ABB RAPID module: 3c2a8035.mod

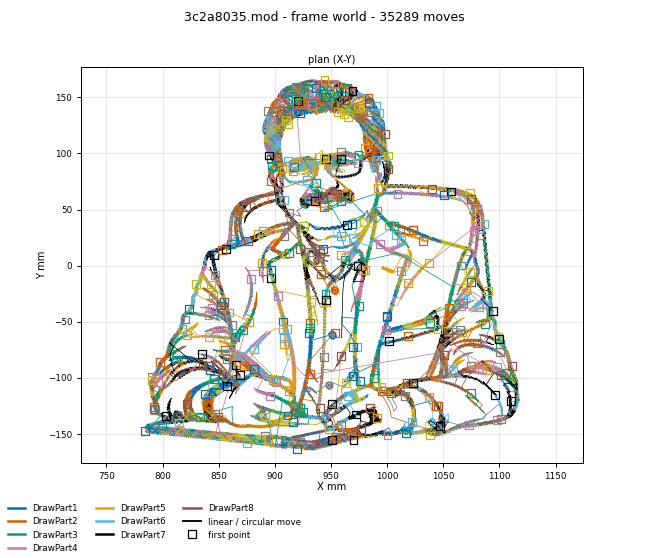
[picture p0: tool path of 3c2a8035.mod in frame world, 35289 of 35291 moves have a stored position in this frame; points joined in program order, loops and branches not executed]
MODULE ImageDraw
  ! Generated 2026-10-07 06:23 for ABB IRB 1600-10/1.45: 2961 strokes
  ! Page 500 x 350 mm. Work object wPaper: Z points up, so pen-up is +Z and the tool uses orientation [0,1,0,0].
  PERS tooldata tPen:=[TRUE,[[0,0,120],[1,0,0,0]],[0.3,[0,0,60],[1,0,0,0],0,0,0]];
  PERS wobjdata wPaper:=[FALSE,TRUE,"",[[700,-175,0],[1,0,0,0]],[[0,0,0],[1,0,0,0]]];
  CONST robtarget pOrigin:=[[0,0,0],[0,1,0,0],[0,0,0,0],[9E9,9E9,9E9,9E9,9E9,9E9]];
  CONST jointtarget jHome:=[[0,0,0,0,30,0],[9E9,9E9,9E9,9E9,9E9,9E9]];
  CONST speeddata vTravel:=[250,200,5000,1000];

  PROC DrawImage()
    SingArea\Wrist;
    ConfL\Off;
    ConfJ\Off;
    MoveAbsJ jHome\NoEOffs,vTravel,fine,tPen;
    DrawPart1;
    DrawPart2;
    DrawPart3;
    DrawPart4;
    DrawPart5;
    DrawPart6;
    DrawPart7;
    DrawPart8;
    DrawPart9;
    DrawPart10;
    DrawPart11;
    DrawPart12;
    DrawPart13;
    DrawPart14;
    DrawPart15;
    DrawPart16;
    DrawPart17;
    DrawPart18;
    DrawPart19;
    DrawPart20;
    DrawPart21;
    DrawPart22;
    DrawPart23;
    DrawPart24;
    DrawPart25;
    DrawPart26;
    DrawPart27;
    DrawPart28;
    DrawPart29;
    DrawPart30;
    DrawPart31;
    DrawPart32;
    DrawPart33;
    DrawPart34;
    DrawPart35;
    DrawPart36;
    DrawPart37;
    DrawPart38;
    DrawPart39;
    DrawPart40;
    DrawPart41;
    DrawPart42;
    DrawPart43;
    DrawPart44;
    DrawPart45;
    DrawPart46;
    DrawPart47;
    DrawPart48;
    DrawPart49;
    DrawPart50;
    DrawPart51;
    DrawPart52;
    DrawPart53;
    DrawPart54;
    DrawPart55;
    DrawPart56;
    DrawPart57;
    DrawPart58;
    DrawPart59;
    DrawPart60;
    DrawPart61;
    DrawPart62;
    DrawPart63;
    DrawPart64;
    DrawPart65;
    DrawPart66;
    DrawPart67;
    DrawPart68;
    DrawPart69;
    DrawPart70;
    DrawPart71;
    DrawPart72;
    DrawPart73;
    DrawPart74;
    DrawPart75;
    DrawPart76;
    DrawPart77;
    DrawPart78;
    DrawPart79;
    DrawPart80;
    DrawPart81;
    DrawPart82;
    DrawPart83;
    DrawPart84;
    DrawPart85;
    DrawPart86;
    DrawPart87;
    DrawPart88;
    DrawPart89;
    DrawPart90;
    DrawPart91;
    DrawPart92;
    DrawPart93;
    DrawPart94;
    DrawPart95;
    DrawPart96;
    DrawPart97;
    DrawPart98;
    DrawPart99;
    DrawPart100;
    DrawPart101;
    DrawPart102;
    DrawPart103;
    DrawPart104;
    DrawPart105;
    DrawPart106;
    DrawPart107;
    DrawPart108;
    DrawPart109;
    DrawPart110;
    DrawPart111;
    DrawPart112;
    DrawPart113;
    DrawPart114;
    DrawPart115;
    DrawPart116;
    DrawPart117;
    DrawPart118;
    DrawPart119;
    DrawPart120;
    DrawPart121;
    DrawPart122;
    DrawPart123;
    DrawPart124;
    DrawPart125;
    DrawPart126;
    DrawPart127;
    DrawPart128;
    DrawPart129;
    DrawPart130;
    DrawPart131;
    DrawPart132;
    DrawPart133;
    DrawPart134;
    DrawPart135;
    DrawPart136;
    DrawPart137;
    DrawPart138;
    DrawPart139;
    DrawPart140;
    DrawPart141;
    DrawPart142;
    DrawPart143;
    DrawPart144;
    DrawPart145;
    DrawPart146;
    DrawPart147;
    DrawPart148;
    DrawPart149;
    DrawPart150;
    DrawPart151;
    DrawPart152;
    DrawPart153;
    DrawPart154;
    DrawPart155;
    DrawPart156;
    DrawPart157;
    DrawPart158;
    DrawPart159;
    DrawPart160;
    DrawPart161;
    DrawPart162;
    DrawPart163;
    DrawPart164;
    DrawPart165;
    DrawPart166;
    DrawPart167;
    DrawPart168;
    DrawPart169;
    DrawPart170;
    DrawPart171;
    DrawPart172;
    DrawPart173;
    DrawPart174;
    DrawPart175;
    DrawPart176;
    DrawPart177;
    DrawPart178;
    DrawPart179;
    DrawPart180;
    DrawPart181;
    DrawPart182;
    DrawPart183;
    DrawPart184;
    DrawPart185;
    DrawPart186;
    DrawPart187;
    DrawPart188;
    DrawPart189;
    DrawPart190;
    DrawPart191;
    DrawPart192;
    DrawPart193;
    DrawPart194;
    DrawPart195;
    DrawPart196;
    DrawPart197;
    DrawPart198;
    DrawPart199;
    DrawPart200;
    DrawPart201;
    DrawPart202;
    DrawPart203;
    DrawPart204;
    DrawPart205;
    DrawPart206;
    DrawPart207;
    DrawPart208;
    DrawPart209;
    DrawPart210;
    DrawPart211;
    DrawPart212;
    DrawPart213;
    DrawPart214;
    DrawPart215;
    DrawPart216;
    DrawPart217;
    DrawPart218;
    DrawPart219;
    DrawPart220;
    DrawPart221;
    DrawPart222;
    DrawPart223;
    DrawPart224;
    DrawPart225;
    DrawPart226;
    DrawPart227;
    DrawPart228;
    DrawPart229;
    DrawPart230;
    DrawPart231;
    DrawPart232;
    DrawPart233;
    DrawPart234;
    DrawPart235;
    DrawPart236;
    DrawPart237;
    DrawPart238;
    DrawPart239;
    DrawPart240;
    DrawPart241;
    DrawPart242;
    DrawPart243;
    DrawPart244;
    DrawPart245;
    DrawPart246;
    DrawPart247;
    DrawPart248;
    DrawPart249;
    DrawPart250;
    DrawPart251;
    DrawPart252;
    DrawPart253;
    DrawPart254;
    DrawPart255;
    DrawPart256;
    DrawPart257;
    DrawPart258;
    DrawPart259;
    DrawPart260;
    DrawPart261;
    DrawPart262;
    DrawPart263;
    DrawPart264;
    DrawPart265;
    DrawPart266;
    DrawPart267;
    DrawPart268;
    DrawPart269;
    DrawPart270;
    DrawPart271;
    DrawPart272;
    DrawPart273;
    DrawPart274;
    DrawPart275;
    DrawPart276;
    DrawPart277;
    DrawPart278;
    DrawPart279;
    DrawPart280;
    DrawPart281;
    DrawPart282;
    DrawPart283;
    DrawPart284;
    DrawPart285;
    DrawPart286;
    DrawPart287;
    DrawPart288;
    DrawPart289;
    DrawPart290;
    DrawPart291;
    DrawPart292;
    DrawPart293;
    DrawPart294;
    DrawPart295;
    MoveAbsJ jHome\NoEOffs,vTravel,fine,tPen;
  ENDPROC

  PROC DrawPart1()
    MoveL Offs(pOrigin,84.39,27.87,6.00),vTravel,z5,tPen\WObj:=wPaper;
    MoveL Offs(pOrigin,84.39,27.87,0.00),v60,z0,tPen\WObj:=wPaper;
    MoveL Offs(pOrigin,86.34,25.92,0.00),v40,z0,tPen\WObj:=wPaper;
    MoveL Offs(pOrigin,86.59,26.62,0.00),v40,z0,tPen\WObj:=wPaper;
    MoveL Offs(pOrigin,99.12,26.62,0.00),v40,fine,tPen\WObj:=wPaper;
    MoveL Offs(pOrigin,99.12,26.62,6.00),v60,z5,tPen\WObj:=wPaper;
    MoveL Offs(pOrigin,99.50,25.13,6.00),vTravel,z5,tPen\WObj:=wPaper;
    MoveL Offs(pOrigin,99.50,25.13,0.00),v60,z0,tPen\WObj:=wPaper;
    MoveL Offs(pOrigin,105.21,30.84,0.00),v40,z0,tPen\WObj:=wPaper;
    MoveL Offs(pOrigin,104.60,31.55,0.00),v40,z0,tPen\WObj:=wPaper;
    MoveL Offs(pOrigin,113.01,23.14,0.00),v40,z0,tPen\WObj:=wPaper;
    MoveL Offs(pOrigin,113.13,23.82,0.00),v40,z0,tPen\WObj:=wPaper;
    MoveL Offs(pOrigin,118.84,29.53,0.00),v40,z0,tPen\WObj:=wPaper;
    MoveL Offs(pOrigin,119.58,30.01,0.00),v40,z0,tPen\WObj:=wPaper;
    MoveL Offs(pOrigin,128.15,21.44,0.00),v40,z0,tPen\WObj:=wPaper;
    MoveL Offs(pOrigin,127.96,22.22,0.00),v40,z0,tPen\WObj:=wPaper;
    MoveL Offs(pOrigin,129.76,24.02,0.00),v40,z0,tPen\WObj:=wPaper;
    MoveL Offs(pOrigin,129.72,23.45,0.00),v40,z0,tPen\WObj:=wPaper;
    MoveL Offs(pOrigin,117.19,23.45,0.00),v40,z0,tPen\WObj:=wPaper;
    MoveL Offs(pOrigin,117.17,23.38,0.00),v40,z0,tPen\WObj:=wPaper;
    MoveL Offs(pOrigin,118.98,25.19,0.00),v40,z0,tPen\WObj:=wPaper;
    MoveL Offs(pOrigin,119.74,24.50,0.00),v40,z0,tPen\WObj:=wPaper;
    MoveL Offs(pOrigin,107.62,24.50,0.00),v40,z0,tPen\WObj:=wPaper;
    MoveL Offs(pOrigin,107.74,24.40,0.00),v40,z0,tPen\WObj:=wPaper;
    MoveL Offs(pOrigin,113.30,29.96,0.00),v40,z0,tPen\WObj:=wPaper;
    MoveL Offs(pOrigin,112.99,30.63,0.00),v40,z0,tPen\WObj:=wPaper;
    MoveL Offs(pOrigin,121.40,22.21,0.00),v40,z0,tPen\WObj:=wPaper;
    MoveL Offs(pOrigin,121.07,22.80,0.00),v40,z0,tPen\WObj:=wPaper;
    MoveL Offs(pOrigin,126.93,28.66,0.00),v40,z0,tPen\WObj:=wPaper;
    MoveL Offs(pOrigin,126.18,29.39,0.00),v40,z0,tPen\WObj:=wPaper;
    MoveL Offs(pOrigin,134.74,20.82,0.00),v40,z0,tPen\WObj:=wPaper;
    MoveL Offs(pOrigin,134.70,21.49,0.00),v40,z0,tPen\WObj:=wPaper;
    MoveL Offs(pOrigin,136.50,23.29,0.00),v40,z0,tPen\WObj:=wPaper;
    MoveL Offs(pOrigin,135.90,24.19,0.00),v40,z0,tPen\WObj:=wPaper;
    MoveL Offs(pOrigin,139.21,27.50,0.00),v40,z0,tPen\WObj:=wPaper;
    MoveL Offs(pOrigin,139.36,28.15,0.00),v40,z0,tPen\WObj:=wPaper;
    MoveL Offs(pOrigin,148.08,19.43,0.00),v40,z0,tPen\WObj:=wPaper;
    MoveL Offs(pOrigin,148.32,20.18,0.00),v40,z0,tPen\WObj:=wPaper;
    MoveL Offs(pOrigin,150.13,21.99,0.00),v40,z0,tPen\WObj:=wPaper;
    MoveL Offs(pOrigin,150.55,21.34,0.00),v40,z0,tPen\WObj:=wPaper;
    MoveL Offs(pOrigin,138.65,21.34,0.00),v40,z0,tPen\WObj:=wPaper;
    MoveL Offs(pOrigin,138.89,21.20,0.00),v40,z0,tPen\WObj:=wPaper;
    MoveL Offs(pOrigin,140.54,22.86,0.00),v40,z0,tPen\WObj:=wPaper;
    MoveL Offs(pOrigin,139.95,23.75,0.00),v40,z0,tPen\WObj:=wPaper;
    MoveL Offs(pOrigin,141.75,25.56,0.00),v40,z0,tPen\WObj:=wPaper;
    MoveL Offs(pOrigin,142.50,26.31,0.00),v40,z0,tPen\WObj:=wPaper;
    MoveL Offs(pOrigin,143.25,27.06,0.00),v40,z0,tPen\WObj:=wPaper;
    MoveL Offs(pOrigin,142.81,27.69,0.00),v40,z0,tPen\WObj:=wPaper;
    MoveL Offs(pOrigin,151.37,19.12,0.00),v40,z0,tPen\WObj:=wPaper;
    MoveL Offs(pOrigin,151.02,19.89,0.00),v40,z0,tPen\WObj:=wPaper;
    MoveL Offs(pOrigin,157.03,25.90,0.00),v40,z0,tPen\WObj:=wPaper;
    MoveL Offs(pOrigin,157.49,26.45,0.00),v40,z0,tPen\WObj:=wPaper;
    MoveL Offs(pOrigin,166.51,17.43,0.00),v40,z0,tPen\WObj:=wPaper;
    MoveL Offs(pOrigin,167.04,17.99,0.00),v40,z0,tPen\WObj:=wPaper;
    MoveL Offs(pOrigin,171.10,22.05,0.00),v40,z0,tPen\WObj:=wPaper;
    MoveL Offs(pOrigin,171.80,21.34,0.00),v40,z0,tPen\WObj:=wPaper;
    MoveL Offs(pOrigin,168.19,21.34,0.00),v40,z0,tPen\WObj:=wPaper;
    MoveL Offs(pOrigin,168.25,22.19,0.00),v40,z0,tPen\WObj:=wPaper;
    MoveL Offs(pOrigin,164.50,18.43,0.00),v40,z0,tPen\WObj:=wPaper;
    MoveL Offs(pOrigin,164.86,17.58,0.00),v40,z0,tPen\WObj:=wPaper;
    MoveL Offs(pOrigin,155.84,26.60,0.00),v40,z0,tPen\WObj:=wPaper;
    MoveL Offs(pOrigin,155.83,26.20,0.00),v40,z0,tPen\WObj:=wPaper;
    MoveL Offs(pOrigin,152.07,22.44,0.00),v40,z0,tPen\WObj:=wPaper;
    MoveL Offs(pOrigin,151.32,21.69,0.00),v40,z0,tPen\WObj:=wPaper;
    MoveL Offs(pOrigin,149.52,19.89,0.00),v40,z0,tPen\WObj:=wPaper;
    MoveL Offs(pOrigin,149.57,19.43,0.00),v40,z0,tPen\WObj:=wPaper;
    MoveL Offs(pOrigin,141.01,27.99,0.00),v40,z0,tPen\WObj:=wPaper;
    MoveL Offs(pOrigin,140.56,27.35,0.00),v40,z0,tPen\WObj:=wPaper;
    MoveL Offs(pOrigin,137.40,24.19,0.00),v40,z0,tPen\WObj:=wPaper;
    MoveL Offs(pOrigin,137.85,23.15,0.00),v40,z0,tPen\WObj:=wPaper;
    MoveL Offs(pOrigin,136.04,21.34,0.00),v40,z0,tPen\WObj:=wPaper;
    MoveL Offs(pOrigin,136.39,20.67,0.00),v40,z0,tPen\WObj:=wPaper;
    MoveL Offs(pOrigin,127.82,29.23,0.00),v40,z0,tPen\WObj:=wPaper;
    MoveL Offs(pOrigin,128.28,28.51,0.00),v40,z0,tPen\WObj:=wPaper;
    MoveL Offs(pOrigin,122.57,22.80,0.00),v40,z0,tPen\WObj:=wPaper;
    MoveL Offs(pOrigin,123.05,22.06,0.00),v40,z0,tPen\WObj:=wPaper;
    MoveL Offs(pOrigin,114.64,30.47,0.00),v40,z0,tPen\WObj:=wPaper;
    MoveL Offs(pOrigin,114.65,29.82,0.00),v40,z0,tPen\WObj:=wPaper;
    MoveL Offs(pOrigin,109.09,24.26,0.00),v40,fine,tPen\WObj:=wPaper;
    MoveL Offs(pOrigin,109.09,24.26,6.00),v60,z5,tPen\WObj:=wPaper;
    MoveL Offs(pOrigin,108.07,23.60,6.00),vTravel,z5,tPen\WObj:=wPaper;
    MoveL Offs(pOrigin,108.07,23.60,0.00),v60,z0,tPen\WObj:=wPaper;
    MoveL Offs(pOrigin,99.80,31.87,0.00),v40,z0,tPen\WObj:=wPaper;
    MoveL Offs(pOrigin,99.67,31.27,0.00),v40,z0,tPen\WObj:=wPaper;
    MoveL Offs(pOrigin,94.11,25.71,0.00),v40,z0,tPen\WObj:=wPaper;
    MoveL Offs(pOrigin,94.88,24.84,0.00),v40,z0,tPen\WObj:=wPaper;
    MoveL Offs(pOrigin,86.02,33.71,0.00),v40,z0,tPen\WObj:=wPaper;
    MoveL Offs(pOrigin,86.59,32.95,0.00),v40,z0,tPen\WObj:=wPaper;
    MoveL Offs(pOrigin,91.05,32.95,0.00),v40,z0,tPen\WObj:=wPaper;
    MoveL Offs(pOrigin,91.89,32.44,0.00),v40,z0,tPen\WObj:=wPaper;
    MoveL Offs(pOrigin,86.18,26.73,0.00),v40,z0,tPen\WObj:=wPaper;
    MoveL Offs(pOrigin,85.74,26.67,0.00),v40,z0,tPen\WObj:=wPaper;
    MoveL Offs(pOrigin,85.31,27.10,0.00),v40,z0,tPen\WObj:=wPaper;
    MoveL Offs(pOrigin,85.74,26.67,0.00),v40,z0,tPen\WObj:=wPaper;
    MoveL Offs(pOrigin,85.28,27.33,0.00),v40,z0,tPen\WObj:=wPaper;
    MoveL Offs(pOrigin,93.39,35.44,0.00),v40,z0,tPen\WObj:=wPaper;
    MoveL Offs(pOrigin,92.90,35.78,0.00),v40,z0,tPen\WObj:=wPaper;
    MoveL Offs(pOrigin,95.30,33.38,0.00),v40,z0,tPen\WObj:=wPaper;
    MoveL Offs(pOrigin,95.04,34.10,0.00),v40,z0,tPen\WObj:=wPaper;
    MoveL Offs(pOrigin,97.29,36.35,0.00),v40,z0,tPen\WObj:=wPaper;
    MoveL Offs(pOrigin,97.84,36.82,0.00),v40,z0,tPen\WObj:=wPaper;
    MoveL Offs(pOrigin,101.15,33.51,0.00),v40,fine,tPen\WObj:=wPaper;
    MoveL Offs(pOrigin,101.15,33.51,6.00),v60,z5,tPen\WObj:=wPaper;
    MoveL Offs(pOrigin,102.34,33.81,6.00),vTravel,z5,tPen\WObj:=wPaper;
    MoveL Offs(pOrigin,102.34,33.81,0.00),v60,z0,tPen\WObj:=wPaper;
    MoveL Offs(pOrigin,98.89,37.26,0.00),v40,z0,tPen\WObj:=wPaper;
    MoveL Offs(pOrigin,99.39,36.96,0.00),v40,z0,tPen\WObj:=wPaper;
    MoveL Offs(pOrigin,96.99,34.56,0.00),v40,z0,tPen\WObj:=wPaper;
    MoveL Offs(pOrigin,96.65,33.52,0.00),v40,z0,tPen\WObj:=wPaper;
    MoveL Offs(pOrigin,94.25,35.93,0.00),v40,z0,tPen\WObj:=wPaper;
    MoveL Offs(pOrigin,94.24,35.06,0.00),v40,z0,tPen\WObj:=wPaper;
    MoveL Offs(pOrigin,98.28,35.06,0.00),v40,z0,tPen\WObj:=wPaper;
    MoveL Offs(pOrigin,98.63,34.71,0.00),v40,z0,tPen\WObj:=wPaper;
    MoveL Offs(pOrigin,101.34,37.42,0.00),v40,z0,tPen\WObj:=wPaper;
    MoveL Offs(pOrigin,101.28,37.85,0.00),v40,z0,tPen\WObj:=wPaper;
    MoveL Offs(pOrigin,105.19,33.95,0.00),v40,fine,tPen\WObj:=wPaper;
    MoveL Offs(pOrigin,105.19,33.95,6.00),v60,z5,tPen\WObj:=wPaper;
    MoveL Offs(pOrigin,106.39,34.24,6.00),vTravel,z5,tPen\WObj:=wPaper;
    MoveL Offs(pOrigin,106.39,34.24,0.00),v60,z0,tPen\WObj:=wPaper;
    MoveL Offs(pOrigin,91.51,49.12,0.00),v40,z0,tPen\WObj:=wPaper;
  ENDPROC

  PROC DrawPart2()
    MoveL Offs(pOrigin,91.94,48.92,0.00),v40,z0,tPen\WObj:=wPaper;
    MoveL Offs(pOrigin,94.79,51.78,0.00),v40,z0,tPen\WObj:=wPaper;
    MoveL Offs(pOrigin,94.45,51.96,0.00),v40,z0,tPen\WObj:=wPaper;
    MoveL Offs(pOrigin,92.32,51.96,0.00),v40,z0,tPen\WObj:=wPaper;
    MoveL Offs(pOrigin,91.95,51.92,0.00),v40,z0,tPen\WObj:=wPaper;
    MoveL Offs(pOrigin,96.30,56.27,0.00),v40,z0,tPen\WObj:=wPaper;
    MoveL Offs(pOrigin,95.94,56.21,0.00),v40,z0,tPen\WObj:=wPaper;
    MoveL Offs(pOrigin,96.43,57.91,0.00),v40,z0,tPen\WObj:=wPaper;
    MoveL Offs(pOrigin,97.35,58.76,0.00),v40,z0,tPen\WObj:=wPaper;
    MoveL Offs(pOrigin,97.35,59.83,0.00),v40,z0,tPen\WObj:=wPaper;
    MoveL Offs(pOrigin,99.20,63.44,0.00),v40,z0,tPen\WObj:=wPaper;
    MoveL Offs(pOrigin,100.12,64.07,0.00),v40,z0,tPen\WObj:=wPaper;
    MoveL Offs(pOrigin,100.40,65.56,0.00),v40,z0,tPen\WObj:=wPaper;
    MoveL Offs(pOrigin,100.40,65.56,0.00),v40,z0,tPen\WObj:=wPaper;
    MoveL Offs(pOrigin,100.40,66.41,0.00),v40,z0,tPen\WObj:=wPaper;
    MoveL Offs(pOrigin,101.32,68.75,0.00),v40,z0,tPen\WObj:=wPaper;
    MoveL Offs(pOrigin,103.94,73.85,0.00),v40,z0,tPen\WObj:=wPaper;
    MoveL Offs(pOrigin,108.69,80.44,0.00),v40,z0,tPen\WObj:=wPaper;
    MoveL Offs(pOrigin,111.88,83.62,0.00),v40,z0,tPen\WObj:=wPaper;
    MoveL Offs(pOrigin,115.70,86.46,0.00),v40,z0,tPen\WObj:=wPaper;
    MoveL Offs(pOrigin,118.25,87.73,0.00),v40,z0,tPen\WObj:=wPaper;
    MoveL Offs(pOrigin,118.75,88.44,0.00),v40,z0,tPen\WObj:=wPaper;
    MoveL Offs(pOrigin,121.86,89.57,0.00),v40,z0,tPen\WObj:=wPaper;
    MoveL Offs(pOrigin,124.84,90.00,0.00),v40,z0,tPen\WObj:=wPaper;
    MoveL Offs(pOrigin,124.84,90.00,0.00),v40,z0,tPen\WObj:=wPaper;
    MoveL Offs(pOrigin,126.96,90.21,0.00),v40,z0,tPen\WObj:=wPaper;
    MoveL Offs(pOrigin,127.18,90.00,0.00),v40,z0,tPen\WObj:=wPaper;
    MoveL Offs(pOrigin,127.18,90.00,0.00),v40,z0,tPen\WObj:=wPaper;
    MoveL Offs(pOrigin,126.54,89.36,0.00),v40,z0,tPen\WObj:=wPaper;
    MoveL Offs(pOrigin,124.84,89.36,0.00),v40,z0,tPen\WObj:=wPaper;
    MoveL Offs(pOrigin,124.84,89.36,0.00),v40,z0,tPen\WObj:=wPaper;
    MoveL Offs(pOrigin,118.46,87.66,0.00),v40,z0,tPen\WObj:=wPaper;
    MoveL Offs(pOrigin,118.12,87.05,0.00),v40,z0,tPen\WObj:=wPaper;
    MoveL Offs(pOrigin,120.82,89.76,0.00),v40,z0,tPen\WObj:=wPaper;
    MoveL Offs(pOrigin,120.75,90.07,0.00),v40,z0,tPen\WObj:=wPaper;
    MoveL Offs(pOrigin,122.85,87.97,0.00),v40,z0,tPen\WObj:=wPaper;
    MoveL Offs(pOrigin,122.62,88.56,0.00),v40,z0,tPen\WObj:=wPaper;
    MoveL Offs(pOrigin,127.13,93.07,0.00),v40,z0,tPen\WObj:=wPaper;
    MoveL Offs(pOrigin,127.63,93.65,0.00),v40,z0,tPen\WObj:=wPaper;
    MoveL Offs(pOrigin,140.10,81.18,0.00),v40,z0,tPen\WObj:=wPaper;
    MoveL Offs(pOrigin,139.82,81.87,0.00),v40,z0,tPen\WObj:=wPaper;
    MoveL Offs(pOrigin,143.13,85.18,0.00),v40,z0,tPen\WObj:=wPaper;
    MoveL Offs(pOrigin,142.69,84.70,0.00),v40,z0,tPen\WObj:=wPaper;
    MoveL Offs(pOrigin,138.65,84.70,0.00),v40,z0,tPen\WObj:=wPaper;
    MoveL Offs(pOrigin,139.07,85.32,0.00),v40,z0,tPen\WObj:=wPaper;
    MoveL Offs(pOrigin,139.50,84.47,0.00),v40,z0,tPen\WObj:=wPaper;
    MoveL Offs(pOrigin,140.77,83.84,0.00),v40,z0,tPen\WObj:=wPaper;
    MoveL Offs(pOrigin,140.99,83.41,0.00),v40,z0,tPen\WObj:=wPaper;
    MoveL Offs(pOrigin,140.99,83.41,0.00),v40,z0,tPen\WObj:=wPaper;
    MoveL Offs(pOrigin,140.35,83.20,0.00),v40,z0,tPen\WObj:=wPaper;
    MoveL Offs(pOrigin,132.91,84.26,0.00),v40,z0,tPen\WObj:=wPaper;
    MoveL Offs(pOrigin,126.96,84.05,0.00),v40,z0,tPen\WObj:=wPaper;
    MoveL Offs(pOrigin,121.65,82.99,0.00),v40,z0,tPen\WObj:=wPaper;
    MoveL Offs(pOrigin,117.40,81.29,0.00),v40,z0,tPen\WObj:=wPaper;
    MoveL Offs(pOrigin,117.26,80.86,0.00),v40,z0,tPen\WObj:=wPaper;
    MoveL Offs(pOrigin,117.82,80.65,0.00),v40,z0,tPen\WObj:=wPaper;
    MoveL Offs(pOrigin,123.78,82.56,0.00),v40,z0,tPen\WObj:=wPaper;
    MoveL Offs(pOrigin,125.26,82.78,0.00),v40,z0,tPen\WObj:=wPaper;
    MoveL Offs(pOrigin,125.90,82.35,0.00),v40,z0,tPen\WObj:=wPaper;
    MoveL Offs(pOrigin,125.90,82.35,0.00),v40,z0,tPen\WObj:=wPaper;
    MoveL Offs(pOrigin,127.60,82.56,0.00),v40,z0,tPen\WObj:=wPaper;
    MoveL Offs(pOrigin,128.24,83.13,0.00),v40,z0,tPen\WObj:=wPaper;
    MoveL Offs(pOrigin,128.88,83.20,0.00),v40,z0,tPen\WObj:=wPaper;
    MoveL Offs(pOrigin,128.02,82.56,0.00),v40,z0,tPen\WObj:=wPaper;
    MoveL Offs(pOrigin,129.09,82.35,0.00),v40,z0,tPen\WObj:=wPaper;
    MoveL Offs(pOrigin,132.27,82.99,0.00),v40,z0,tPen\WObj:=wPaper;
    MoveL Offs(pOrigin,135.04,82.99,0.00),v40,z0,tPen\WObj:=wPaper;
    MoveL Offs(pOrigin,142.90,81.50,0.00),v40,z0,tPen\WObj:=wPaper;
    MoveL Offs(pOrigin,163.30,74.77,0.00),v40,z0,tPen\WObj:=wPaper;
    MoveL Offs(pOrigin,169.39,72.08,0.00),v40,z0,tPen\WObj:=wPaper;
    MoveL Offs(pOrigin,169.53,71.51,0.00),v40,z0,tPen\WObj:=wPaper;
    MoveL Offs(pOrigin,169.04,70.95,0.00),v40,z0,tPen\WObj:=wPaper;
    MoveL Offs(pOrigin,168.61,70.95,0.00),v40,z0,tPen\WObj:=wPaper;
    MoveL Offs(pOrigin,164.79,73.28,0.00),v40,z0,tPen\WObj:=wPaper;
    MoveL Offs(pOrigin,159.48,74.91,0.00),v40,z0,tPen\WObj:=wPaper;
    MoveL Offs(pOrigin,152.25,75.12,0.00),v40,z0,tPen\WObj:=wPaper;
    MoveL Offs(pOrigin,146.30,73.85,0.00),v40,z0,tPen\WObj:=wPaper;
    MoveL Offs(pOrigin,142.69,72.65,0.00),v40,z0,tPen\WObj:=wPaper;
    MoveL Offs(pOrigin,130.79,67.33,0.00),v40,z0,tPen\WObj:=wPaper;
    MoveL Offs(pOrigin,124.20,63.01,0.00),v40,z0,tPen\WObj:=wPaper;
    MoveL Offs(pOrigin,122.00,60.46,0.00),v40,z0,tPen\WObj:=wPaper;
    MoveL Offs(pOrigin,119.95,54.51,0.00),v40,z0,tPen\WObj:=wPaper;
    MoveL Offs(pOrigin,119.31,49.41,0.00),v40,z0,tPen\WObj:=wPaper;
    MoveL Offs(pOrigin,119.74,43.46,0.00),v40,z0,tPen\WObj:=wPaper;
    MoveL Offs(pOrigin,120.52,40.06,0.00),v40,z0,tPen\WObj:=wPaper;
    MoveL Offs(pOrigin,118.68,39.71,0.00),v40,z0,tPen\WObj:=wPaper;
    MoveL Offs(pOrigin,117.75,41.97,0.00),v40,z0,tPen\WObj:=wPaper;
    MoveL Offs(pOrigin,116.97,42.40,0.00),v40,z0,tPen\WObj:=wPaper;
    MoveL Offs(pOrigin,116.97,42.40,0.00),v40,z0,tPen\WObj:=wPaper;
    MoveL Offs(pOrigin,117.19,40.91,0.00),v40,z0,tPen\WObj:=wPaper;
    MoveL Offs(pOrigin,116.76,40.63,0.00),v40,z0,tPen\WObj:=wPaper;
    MoveL Offs(pOrigin,115.84,42.19,0.00),v40,z0,tPen\WObj:=wPaper;
    MoveL Offs(pOrigin,115.70,43.46,0.00),v40,z0,tPen\WObj:=wPaper;
    MoveL Offs(pOrigin,115.70,43.51,0.00),v40,z0,tPen\WObj:=wPaper;
    MoveL Offs(pOrigin,113.58,43.51,0.00),v40,z0,tPen\WObj:=wPaper;
    MoveL Offs(pOrigin,113.57,44.31,0.00),v40,z0,tPen\WObj:=wPaper;
    MoveL Offs(pOrigin,114.43,40.91,0.00),v40,z0,tPen\WObj:=wPaper;
    MoveL Offs(pOrigin,115.06,40.91,0.00),v40,z0,tPen\WObj:=wPaper;
    MoveL Offs(pOrigin,114.85,42.61,0.00),v40,z0,tPen\WObj:=wPaper;
    MoveL Offs(pOrigin,115.28,43.46,0.00),v40,z0,tPen\WObj:=wPaper;
    MoveL Offs(pOrigin,115.28,43.46,0.00),v40,z0,tPen\WObj:=wPaper;
    MoveL Offs(pOrigin,114.85,44.74,0.00),v40,z0,tPen\WObj:=wPaper;
    MoveL Offs(pOrigin,114.99,45.10,0.00),v40,z0,tPen\WObj:=wPaper;
    MoveL Offs(pOrigin,106.43,36.53,0.00),v40,fine,tPen\WObj:=wPaper;
    MoveL Offs(pOrigin,106.43,36.53,6.00),v60,z5,tPen\WObj:=wPaper;
    MoveL Offs(pOrigin,108.08,36.69,6.00),vTravel,z5,tPen\WObj:=wPaper;
    MoveL Offs(pOrigin,108.08,36.69,0.00),v60,z0,tPen\WObj:=wPaper;
    MoveL Offs(pOrigin,116.04,44.65,0.00),v40,z0,tPen\WObj:=wPaper;
    MoveL Offs(pOrigin,116.39,45.15,0.00),v40,z0,tPen\WObj:=wPaper;
    MoveL Offs(pOrigin,117.44,44.10,0.00),v40,z0,tPen\WObj:=wPaper;
    MoveL Offs(pOrigin,116.64,43.75,0.00),v40,z0,tPen\WObj:=wPaper;
    MoveL Offs(pOrigin,109.88,36.99,0.00),v40,z0,tPen\WObj:=wPaper;
    MoveL Offs(pOrigin,110.18,37.18,0.00),v40,z0,tPen\WObj:=wPaper;
    MoveL Offs(pOrigin,103.16,37.18,0.00),v40,z0,tPen\WObj:=wPaper;
    MoveL Offs(pOrigin,103.38,36.12,0.00),v40,z0,tPen\WObj:=wPaper;
    MoveL Offs(pOrigin,98.49,36.12,0.00),v40,fine,tPen\WObj:=wPaper;
    MoveL Offs(pOrigin,98.49,36.12,6.00),v60,z5,tPen\WObj:=wPaper;
    MoveL Offs(pOrigin,96.49,36.67,6.00),vTravel,z5,tPen\WObj:=wPaper;
    MoveL Offs(pOrigin,96.49,36.67,0.00),v60,z0,tPen\WObj:=wPaper;
    MoveL Offs(pOrigin,99.65,33.51,0.00),v40,fine,tPen\WObj:=wPaper;
  ENDPROC

  PROC DrawPart3()
    MoveL Offs(pOrigin,99.65,33.51,6.00),v60,z5,tPen\WObj:=wPaper;
    MoveL Offs(pOrigin,98.15,33.52,6.00),vTravel,z5,tPen\WObj:=wPaper;
    MoveL Offs(pOrigin,98.15,33.52,0.00),v60,z0,tPen\WObj:=wPaper;
    MoveL Offs(pOrigin,95.45,36.22,0.00),v40,z0,tPen\WObj:=wPaper;
    MoveL Offs(pOrigin,95.34,35.90,0.00),v40,z0,tPen\WObj:=wPaper;
    MoveL Offs(pOrigin,92.94,33.49,0.00),v40,z0,tPen\WObj:=wPaper;
    MoveL Offs(pOrigin,93.60,34.01,0.00),v40,z0,tPen\WObj:=wPaper;
    MoveL Offs(pOrigin,90.20,34.01,0.00),v40,z0,tPen\WObj:=wPaper;
    MoveL Offs(pOrigin,89.20,34.23,0.00),v40,z0,tPen\WObj:=wPaper;
    MoveL Offs(pOrigin,84.84,29.87,0.00),v40,z0,tPen\WObj:=wPaper;
    MoveL Offs(pOrigin,85.31,29.78,0.00),v40,z0,tPen\WObj:=wPaper;
    MoveL Offs(pOrigin,87.86,29.78,0.00),v40,z0,tPen\WObj:=wPaper;
    MoveL Offs(pOrigin,88.07,29.23,0.00),v40,z0,tPen\WObj:=wPaper;
    MoveL Offs(pOrigin,106.56,27.52,0.00),v40,z0,tPen\WObj:=wPaper;
    MoveL Offs(pOrigin,192.41,18.60,0.00),v40,z0,tPen\WObj:=wPaper;
    MoveL Offs(pOrigin,192.98,18.32,0.00),v40,z0,tPen\WObj:=wPaper;
    MoveL Offs(pOrigin,193.05,17.33,0.00),v40,z0,tPen\WObj:=wPaper;
    MoveL Offs(pOrigin,192.84,17.11,0.00),v40,z0,tPen\WObj:=wPaper;
    MoveL Offs(pOrigin,188.80,17.33,0.00),v40,z0,tPen\WObj:=wPaper;
    MoveL Offs(pOrigin,148.00,21.79,0.00),v40,z0,tPen\WObj:=wPaper;
    MoveL Offs(pOrigin,87.65,27.74,0.00),v40,z0,tPen\WObj:=wPaper;
    MoveL Offs(pOrigin,86.66,28.02,0.00),v40,z0,tPen\WObj:=wPaper;
    MoveL Offs(pOrigin,86.59,29.01,0.00),v40,z0,tPen\WObj:=wPaper;
    MoveL Offs(pOrigin,88.07,29.23,0.00),v40,z0,tPen\WObj:=wPaper;
    MoveL Offs(pOrigin,87.01,28.73,0.00),v40,z0,tPen\WObj:=wPaper;
    MoveL Offs(pOrigin,85.31,28.73,0.00),v40,z0,tPen\WObj:=wPaper;
    MoveL Offs(pOrigin,85.55,28.38,0.00),v40,z0,tPen\WObj:=wPaper;
    MoveL Offs(pOrigin,85.55,31.14,0.00),v40,z0,tPen\WObj:=wPaper;
    MoveL Offs(pOrigin,85.31,30.84,0.00),v40,z0,tPen\WObj:=wPaper;
    MoveL Offs(pOrigin,87.22,30.84,0.00),v40,z0,tPen\WObj:=wPaper;
    MoveL Offs(pOrigin,86.61,31.56,0.00),v40,z0,tPen\WObj:=wPaper;
    MoveL Offs(pOrigin,86.61,32.62,0.00),v40,z0,tPen\WObj:=wPaper;
    MoveL Offs(pOrigin,85.53,32.62,0.00),v40,z0,tPen\WObj:=wPaper;
    MoveL Offs(pOrigin,85.95,33.05,0.00),v40,z0,tPen\WObj:=wPaper;
    MoveL Offs(pOrigin,85.53,32.62,0.00),v40,z0,tPen\WObj:=wPaper;
    MoveL Offs(pOrigin,85.27,32.96,0.00),v40,z0,tPen\WObj:=wPaper;
    MoveL Offs(pOrigin,93.08,25.15,0.00),v40,z0,tPen\WObj:=wPaper;
    MoveL Offs(pOrigin,92.76,25.85,0.00),v40,z0,tPen\WObj:=wPaper;
    MoveL Offs(pOrigin,98.32,31.41,0.00),v40,z0,tPen\WObj:=wPaper;
    MoveL Offs(pOrigin,98.00,32.17,0.00),v40,z0,tPen\WObj:=wPaper;
    MoveL Offs(pOrigin,106.42,23.76,0.00),v40,z0,tPen\WObj:=wPaper;
    MoveL Offs(pOrigin,106.24,24.40,0.00),v40,z0,tPen\WObj:=wPaper;
    MoveL Offs(pOrigin,112.10,30.26,0.00),v40,z0,tPen\WObj:=wPaper;
    MoveL Offs(pOrigin,111.49,30.63,0.00),v40,z0,tPen\WObj:=wPaper;
    MoveL Offs(pOrigin,119.91,22.22,0.00),v40,z0,tPen\WObj:=wPaper;
    MoveL Offs(pOrigin,119.87,23.09,0.00),v40,z0,tPen\WObj:=wPaper;
    MoveL Offs(pOrigin,121.52,24.74,0.00),v40,z0,tPen\WObj:=wPaper;
    MoveL Offs(pOrigin,122.27,25.50,0.00),v40,z0,tPen\WObj:=wPaper;
    MoveL Offs(pOrigin,125.58,28.80,0.00),v40,fine,tPen\WObj:=wPaper;
    MoveL Offs(pOrigin,125.58,28.80,6.00),v60,z5,tPen\WObj:=wPaper;
    MoveL Offs(pOrigin,124.38,29.69,6.00),vTravel,z5,tPen\WObj:=wPaper;
    MoveL Offs(pOrigin,124.38,29.69,0.00),v60,z0,tPen\WObj:=wPaper;
    MoveL Offs(pOrigin,132.94,21.13,0.00),v40,z0,tPen\WObj:=wPaper;
    MoveL Offs(pOrigin,133.35,21.63,0.00),v40,z0,tPen\WObj:=wPaper;
    MoveL Offs(pOrigin,135.00,23.29,0.00),v40,z0,tPen\WObj:=wPaper;
    MoveL Offs(pOrigin,134.55,24.33,0.00),v40,z0,tPen\WObj:=wPaper;
    MoveL Offs(pOrigin,137.86,27.64,0.00),v40,z0,tPen\WObj:=wPaper;
    MoveL Offs(pOrigin,137.71,28.30,0.00),v40,z0,tPen\WObj:=wPaper;
    MoveL Offs(pOrigin,146.43,19.59,0.00),v40,z0,tPen\WObj:=wPaper;
    MoveL Offs(pOrigin,146.98,20.33,0.00),v40,z0,tPen\WObj:=wPaper;
    MoveL Offs(pOrigin,152.99,26.34,0.00),v40,z0,tPen\WObj:=wPaper;
    MoveL Offs(pOrigin,152.55,26.91,0.00),v40,z0,tPen\WObj:=wPaper;
    MoveL Offs(pOrigin,161.56,17.89,0.00),v40,z0,tPen\WObj:=wPaper;
    MoveL Offs(pOrigin,161.80,18.73,0.00),v40,z0,tPen\WObj:=wPaper;
    MoveL Offs(pOrigin,165.86,22.78,0.00),v40,fine,tPen\WObj:=wPaper;
    MoveL Offs(pOrigin,165.86,22.78,6.00),v60,z5,tPen\WObj:=wPaper;
    MoveL Offs(pOrigin,164.66,23.08,6.00),vTravel,z5,tPen\WObj:=wPaper;
    MoveL Offs(pOrigin,164.66,23.08,0.00),v60,z0,tPen\WObj:=wPaper;
    MoveL Offs(pOrigin,160.45,18.87,0.00),v40,z0,tPen\WObj:=wPaper;
    MoveL Offs(pOrigin,159.92,18.05,0.00),v40,z0,tPen\WObj:=wPaper;
    MoveL Offs(pOrigin,150.90,27.07,0.00),v40,z0,tPen\WObj:=wPaper;
    MoveL Offs(pOrigin,150.29,26.63,0.00),v40,z0,tPen\WObj:=wPaper;
    MoveL Offs(pOrigin,146.83,23.17,0.00),v40,fine,tPen\WObj:=wPaper;
    MoveL Offs(pOrigin,146.83,23.17,6.00),v60,z5,tPen\WObj:=wPaper;
    MoveL Offs(pOrigin,145.93,22.27,6.00),vTravel,z5,tPen\WObj:=wPaper;
    MoveL Offs(pOrigin,145.93,22.27,0.00),v60,z0,tPen\WObj:=wPaper;
    MoveL Offs(pOrigin,144.28,20.62,0.00),v40,z0,tPen\WObj:=wPaper;
    MoveL Offs(pOrigin,144.78,19.74,0.00),v40,z0,tPen\WObj:=wPaper;
    MoveL Offs(pOrigin,135.92,28.61,0.00),v40,z0,tPen\WObj:=wPaper;
    MoveL Offs(pOrigin,136.51,27.79,0.00),v40,z0,tPen\WObj:=wPaper;
    MoveL Offs(pOrigin,133.36,24.63,0.00),v40,z0,tPen\WObj:=wPaper;
    MoveL Offs(pOrigin,133.80,23.58,0.00),v40,z0,tPen\WObj:=wPaper;
    MoveL Offs(pOrigin,132.00,21.78,0.00),v40,z0,tPen\WObj:=wPaper;
    MoveL Offs(pOrigin,131.29,21.28,0.00),v40,z0,tPen\WObj:=wPaper;
    MoveL Offs(pOrigin,122.88,29.70,0.00),v40,z0,tPen\WObj:=wPaper;
    MoveL Offs(pOrigin,123.03,29.24,0.00),v40,z0,tPen\WObj:=wPaper;
    MoveL Offs(pOrigin,119.73,25.94,0.00),v40,fine,tPen\WObj:=wPaper;
    MoveL Offs(pOrigin,119.73,25.94,6.00),v60,z5,tPen\WObj:=wPaper;
    MoveL Offs(pOrigin,118.68,26.62,6.00),vTravel,z5,tPen\WObj:=wPaper;
    MoveL Offs(pOrigin,118.68,26.62,0.00),v60,z0,tPen\WObj:=wPaper;
    MoveL Offs(pOrigin,123.56,26.62,0.00),v40,z0,tPen\WObj:=wPaper;
    MoveL Offs(pOrigin,123.14,27.52,0.00),v40,z0,tPen\WObj:=wPaper;
    MoveL Offs(pOrigin,122.29,28.16,0.00),v40,z0,tPen\WObj:=wPaper;
    MoveL Offs(pOrigin,121.30,27.88,0.00),v40,z0,tPen\WObj:=wPaper;
    MoveL Offs(pOrigin,122.07,26.89,0.00),v40,z0,tPen\WObj:=wPaper;
    MoveL Offs(pOrigin,123.56,27.52,0.00),v40,z0,tPen\WObj:=wPaper;
    MoveL Offs(pOrigin,129.94,27.10,0.00),v40,z0,tPen\WObj:=wPaper;
    MoveL Offs(pOrigin,129.94,27.10,0.00),v40,z0,tPen\WObj:=wPaper;
    MoveL Offs(pOrigin,129.94,28.38,0.00),v40,z0,tPen\WObj:=wPaper;
    MoveL Offs(pOrigin,129.94,28.38,0.00),v40,z0,tPen\WObj:=wPaper;
    MoveL Offs(pOrigin,109.96,30.29,0.00),v40,z0,tPen\WObj:=wPaper;
    MoveL Offs(pOrigin,109.96,30.29,0.00),v40,z0,tPen\WObj:=wPaper;
    MoveL Offs(pOrigin,110.03,29.44,0.00),v40,z0,tPen\WObj:=wPaper;
    MoveL Offs(pOrigin,110.39,29.23,0.00),v40,z0,tPen\WObj:=wPaper;
    MoveL Offs(pOrigin,113.36,29.01,0.00),v40,z0,tPen\WObj:=wPaper;
    MoveL Offs(pOrigin,114.21,28.52,0.00),v40,z0,tPen\WObj:=wPaper;
    MoveL Offs(pOrigin,115.91,28.80,0.00),v40,z0,tPen\WObj:=wPaper;
    MoveL Offs(pOrigin,116.55,28.38,0.00),v40,z0,tPen\WObj:=wPaper;
    MoveL Offs(pOrigin,118.25,28.59,0.00),v40,z0,tPen\WObj:=wPaper;
    MoveL Offs(pOrigin,118.89,28.16,0.00),v40,z0,tPen\WObj:=wPaper;
    MoveL Offs(pOrigin,118.89,28.16,0.00),v40,z0,tPen\WObj:=wPaper;
    MoveL Offs(pOrigin,120.38,28.38,0.00),v40,z0,tPen\WObj:=wPaper;
    MoveL Offs(pOrigin,120.94,27.74,0.00),v40,z0,tPen\WObj:=wPaper;
    MoveL Offs(pOrigin,119.95,27.10,0.00),v40,z0,tPen\WObj:=wPaper;
    MoveL Offs(pOrigin,118.89,27.74,0.00),v40,z0,tPen\WObj:=wPaper;
    MoveL Offs(pOrigin,118.89,27.74,0.00),v40,z0,tPen\WObj:=wPaper;
    MoveL Offs(pOrigin,118.25,27.31,0.00),v40,z0,tPen\WObj:=wPaper;
    MoveL Offs(pOrigin,117.40,27.31,0.00),v40,z0,tPen\WObj:=wPaper;
    MoveL Offs(pOrigin,116.55,28.02,0.00),v40,z0,tPen\WObj:=wPaper;
    MoveL Offs(pOrigin,115.28,27.52,0.00),v40,z0,tPen\WObj:=wPaper;
  ENDPROC

  PROC DrawPart4()
    MoveL Offs(pOrigin,114.43,28.38,0.00),v40,z0,tPen\WObj:=wPaper;
    MoveL Offs(pOrigin,114.00,28.38,0.00),v40,z0,tPen\WObj:=wPaper;
    MoveL Offs(pOrigin,113.36,27.81,0.00),v40,z0,tPen\WObj:=wPaper;
    MoveL Offs(pOrigin,110.18,27.95,0.00),v40,z0,tPen\WObj:=wPaper;
    MoveL Offs(pOrigin,109.32,28.38,0.00),v40,z0,tPen\WObj:=wPaper;
    MoveL Offs(pOrigin,109.32,28.38,0.00),v40,z0,tPen\WObj:=wPaper;
    MoveL Offs(pOrigin,107.84,28.16,0.00),v40,z0,tPen\WObj:=wPaper;
    MoveL Offs(pOrigin,107.41,28.80,0.00),v40,z0,tPen\WObj:=wPaper;
    MoveL Offs(pOrigin,107.41,28.80,0.00),v40,z0,tPen\WObj:=wPaper;
    MoveL Offs(pOrigin,106.14,28.38,0.00),v40,z0,tPen\WObj:=wPaper;
    MoveL Offs(pOrigin,105.07,29.08,0.00),v40,z0,tPen\WObj:=wPaper;
    MoveL Offs(pOrigin,104.22,28.59,0.00),v40,z0,tPen\WObj:=wPaper;
    MoveL Offs(pOrigin,103.38,28.59,0.00),v40,z0,tPen\WObj:=wPaper;
    MoveL Offs(pOrigin,102.53,29.23,0.00),v40,z0,tPen\WObj:=wPaper;
    MoveL Offs(pOrigin,102.53,29.65,0.00),v40,z0,tPen\WObj:=wPaper;
    MoveL Offs(pOrigin,101.89,30.08,0.00),v40,z0,tPen\WObj:=wPaper;
    MoveL Offs(pOrigin,98.06,30.71,0.00),v40,z0,tPen\WObj:=wPaper;
    MoveL Offs(pOrigin,89.78,31.35,0.00),v40,z0,tPen\WObj:=wPaper;
    MoveL Offs(pOrigin,89.14,31.77,0.00),v40,z0,tPen\WObj:=wPaper;
    MoveL Offs(pOrigin,89.14,31.77,0.00),v40,z0,tPen\WObj:=wPaper;
    MoveL Offs(pOrigin,89.14,32.41,0.00),v40,z0,tPen\WObj:=wPaper;
    MoveL Offs(pOrigin,89.78,32.41,0.00),v40,z0,tPen\WObj:=wPaper;
    MoveL Offs(pOrigin,89.78,32.41,0.00),v40,z0,tPen\WObj:=wPaper;
    MoveL Offs(pOrigin,109.96,30.29,0.00),v40,z0,tPen\WObj:=wPaper;
    MoveL Offs(pOrigin,109.84,30.79,0.00),v40,z0,tPen\WObj:=wPaper;
    MoveL Offs(pOrigin,118.11,22.52,0.00),v40,z0,tPen\WObj:=wPaper;
    MoveL Offs(pOrigin,118.37,23.09,0.00),v40,z0,tPen\WObj:=wPaper;
    MoveL Offs(pOrigin,124.08,28.80,0.00),v40,fine,tPen\WObj:=wPaper;
    MoveL Offs(pOrigin,124.08,28.80,6.00),v60,z5,tPen\WObj:=wPaper;
    MoveL Offs(pOrigin,121.54,29.24,6.00),vTravel,z5,tPen\WObj:=wPaper;
    MoveL Offs(pOrigin,121.54,29.24,0.00),v60,z0,tPen\WObj:=wPaper;
    MoveL Offs(pOrigin,118.38,26.08,0.00),v40,z0,tPen\WObj:=wPaper;
    MoveL Offs(pOrigin,117.63,25.33,0.00),v40,z0,tPen\WObj:=wPaper;
    MoveL Offs(pOrigin,115.83,23.53,0.00),v40,z0,tPen\WObj:=wPaper;
    MoveL Offs(pOrigin,116.46,22.68,0.00),v40,z0,tPen\WObj:=wPaper;
    MoveL Offs(pOrigin,108.04,31.09,0.00),v40,z0,tPen\WObj:=wPaper;
    MoveL Offs(pOrigin,108.06,30.70,0.00),v40,z0,tPen\WObj:=wPaper;
    MoveL Offs(pOrigin,102.20,24.83,0.00),v40,z0,tPen\WObj:=wPaper;
    MoveL Offs(pOrigin,101.47,24.22,0.00),v40,z0,tPen\WObj:=wPaper;
    MoveL Offs(pOrigin,90.51,35.19,0.00),v40,z0,tPen\WObj:=wPaper;
    MoveL Offs(pOrigin,91.29,34.84,0.00),v40,z0,tPen\WObj:=wPaper;
    MoveL Offs(pOrigin,84.83,28.38,0.00),v40,z0,tPen\WObj:=wPaper;
    MoveL Offs(pOrigin,85.52,27.67,0.00),v40,z0,tPen\WObj:=wPaper;
    MoveL Offs(pOrigin,88.50,27.67,0.00),v40,fine,tPen\WObj:=wPaper;
    MoveL Offs(pOrigin,88.50,27.67,6.00),v60,z5,tPen\WObj:=wPaper;
    MoveL Offs(pOrigin,88.72,26.29,6.00),vTravel,z5,tPen\WObj:=wPaper;
    MoveL Offs(pOrigin,88.72,26.29,0.00),v60,z0,tPen\WObj:=wPaper;
    MoveL Offs(pOrigin,94.28,31.85,0.00),v40,fine,tPen\WObj:=wPaper;
    MoveL Offs(pOrigin,94.28,31.85,6.00),v60,z5,tPen\WObj:=wPaper;
    MoveL Offs(pOrigin,92.93,32.00,6.00),vTravel,z5,tPen\WObj:=wPaper;
    MoveL Offs(pOrigin,92.93,32.00,0.00),v60,z0,tPen\WObj:=wPaper;
    MoveL Offs(pOrigin,87.22,26.29,0.00),v40,z0,tPen\WObj:=wPaper;
    MoveL Offs(pOrigin,88.14,25.61,0.00),v40,z0,tPen\WObj:=wPaper;
    MoveL Offs(pOrigin,84.38,29.37,0.00),v40,fine,tPen\WObj:=wPaper;
    MoveL Offs(pOrigin,84.38,29.37,6.00),v60,z5,tPen\WObj:=wPaper;
    MoveL Offs(pOrigin,84.38,30.86,6.00),vTravel,z5,tPen\WObj:=wPaper;
    MoveL Offs(pOrigin,84.38,30.86,0.00),v60,z0,tPen\WObj:=wPaper;
    MoveL Offs(pOrigin,89.94,25.30,0.00),v40,z0,tPen\WObj:=wPaper;
    MoveL Offs(pOrigin,89.92,26.00,0.00),v40,z0,tPen\WObj:=wPaper;
    MoveL Offs(pOrigin,95.78,31.86,0.00),v40,z0,tPen\WObj:=wPaper;
    MoveL Offs(pOrigin,96.36,32.33,0.00),v40,z0,tPen\WObj:=wPaper;
    MoveL Offs(pOrigin,104.62,24.06,0.00),v40,z0,tPen\WObj:=wPaper;
    MoveL Offs(pOrigin,105.04,24.69,0.00),v40,z0,tPen\WObj:=wPaper;
    MoveL Offs(pOrigin,110.60,30.25,0.00),v40,fine,tPen\WObj:=wPaper;
    MoveL Offs(pOrigin,110.60,30.25,6.00),v60,z5,tPen\WObj:=wPaper;
    MoveL Offs(pOrigin,109.26,30.40,6.00),vTravel,z5,tPen\WObj:=wPaper;
    MoveL Offs(pOrigin,109.26,30.40,0.00),v60,z0,tPen\WObj:=wPaper;
    MoveL Offs(pOrigin,103.70,24.84,0.00),v40,z0,tPen\WObj:=wPaper;
    MoveL Offs(pOrigin,103.12,24.07,0.00),v40,z0,tPen\WObj:=wPaper;
    MoveL Offs(pOrigin,91.85,35.34,0.00),v40,fine,tPen\WObj:=wPaper;
    MoveL Offs(pOrigin,91.85,35.34,6.00),v60,z5,tPen\WObj:=wPaper;
    MoveL Offs(pOrigin,89.46,34.74,6.00),vTravel,z5,tPen\WObj:=wPaper;
    MoveL Offs(pOrigin,89.46,34.74,0.00),v60,z0,tPen\WObj:=wPaper;
    MoveL Offs(pOrigin,99.68,24.53,0.00),v40,fine,tPen\WObj:=wPaper;
    MoveL Offs(pOrigin,99.68,24.53,6.00),v60,z5,tPen\WObj:=wPaper;
    MoveL Offs(pOrigin,100.85,24.98,6.00),vTravel,z5,tPen\WObj:=wPaper;
    MoveL Offs(pOrigin,100.85,24.98,0.00),v60,z0,tPen\WObj:=wPaper;
    MoveL Offs(pOrigin,106.56,30.69,0.00),v40,z0,tPen\WObj:=wPaper;
    MoveL Offs(pOrigin,106.40,31.25,0.00),v40,z0,tPen\WObj:=wPaper;
    MoveL Offs(pOrigin,114.66,22.98,0.00),v40,z0,tPen\WObj:=wPaper;
    MoveL Offs(pOrigin,114.48,23.67,0.00),v40,z0,tPen\WObj:=wPaper;
    MoveL Offs(pOrigin,120.19,29.38,0.00),v40,fine,tPen\WObj:=wPaper;
    MoveL Offs(pOrigin,120.19,29.38,6.00),v60,z5,tPen\WObj:=wPaper;
    MoveL Offs(pOrigin,121.38,29.70,6.00),vTravel,z5,tPen\WObj:=wPaper;
    MoveL Offs(pOrigin,121.38,29.70,0.00),v60,z0,tPen\WObj:=wPaper;
    MoveL Offs(pOrigin,129.95,21.14,0.00),v40,z0,tPen\WObj:=wPaper;
    MoveL Offs(pOrigin,129.30,22.07,0.00),v40,z0,tPen\WObj:=wPaper;
    MoveL Offs(pOrigin,130.96,23.72,0.00),v40,z0,tPen\WObj:=wPaper;
    MoveL Offs(pOrigin,130.51,24.77,0.00),v40,z0,tPen\WObj:=wPaper;
    MoveL Offs(pOrigin,133.82,28.08,0.00),v40,z0,tPen\WObj:=wPaper;
    MoveL Offs(pOrigin,134.42,28.61,0.00),v40,z0,tPen\WObj:=wPaper;
    MoveL Offs(pOrigin,142.98,20.05,0.00),v40,z0,tPen\WObj:=wPaper;
    MoveL Offs(pOrigin,142.93,20.77,0.00),v40,z0,tPen\WObj:=wPaper;
    MoveL Offs(pOrigin,144.74,22.57,0.00),v40,z0,tPen\WObj:=wPaper;
    MoveL Offs(pOrigin,145.49,23.32,0.00),v40,z0,tPen\WObj:=wPaper;
    MoveL Offs(pOrigin,148.79,26.63,0.00),v40,z0,tPen\WObj:=wPaper;
    MoveL Offs(pOrigin,149.25,27.22,0.00),v40,z0,tPen\WObj:=wPaper;
    MoveL Offs(pOrigin,158.12,18.35,0.00),v40,z0,tPen\WObj:=wPaper;
    MoveL Offs(pOrigin,158.20,19.22,0.00),v40,z0,tPen\WObj:=wPaper;
    MoveL Offs(pOrigin,171.16,19.22,0.00),v40,fine,tPen\WObj:=wPaper;
    MoveL Offs(pOrigin,171.16,19.22,6.00),v60,z5,tPen\WObj:=wPaper;
    MoveL Offs(pOrigin,171.23,17.71,6.00),vTravel,z5,tPen\WObj:=wPaper;
    MoveL Offs(pOrigin,171.23,17.71,0.00),v60,z0,tPen\WObj:=wPaper;
    MoveL Offs(pOrigin,175.14,21.61,0.00),v40,fine,tPen\WObj:=wPaper;
    MoveL Offs(pOrigin,175.14,21.61,6.00),v60,z5,tPen\WObj:=wPaper;
    MoveL Offs(pOrigin,173.94,21.91,6.00),vTravel,z5,tPen\WObj:=wPaper;
    MoveL Offs(pOrigin,173.94,21.91,0.00),v60,z0,tPen\WObj:=wPaper;
    MoveL Offs(pOrigin,169.74,17.70,0.00),v40,z0,tPen\WObj:=wPaper;
    MoveL Offs(pOrigin,169.96,16.97,0.00),v40,z0,tPen\WObj:=wPaper;
    MoveL Offs(pOrigin,160.79,26.14,0.00),v40,z0,tPen\WObj:=wPaper;
    MoveL Offs(pOrigin,161.22,25.62,0.00),v40,z0,tPen\WObj:=wPaper;
    MoveL Offs(pOrigin,160.32,24.71,0.00),v40,z0,tPen\WObj:=wPaper;
    MoveL Offs(pOrigin,159.87,25.76,0.00),v40,z0,tPen\WObj:=wPaper;
    MoveL Offs(pOrigin,158.82,24.71,0.00),v40,z0,tPen\WObj:=wPaper;
    MoveL Offs(pOrigin,157.99,23.91,0.00),v40,z0,tPen\WObj:=wPaper;
    MoveL Offs(pOrigin,156.93,24.55,0.00),v40,z0,tPen\WObj:=wPaper;
    MoveL Offs(pOrigin,156.93,24.55,0.00),v40,z0,tPen\WObj:=wPaper;
    MoveL Offs(pOrigin,157.35,24.98,0.00),v40,z0,tPen\WObj:=wPaper;
    MoveL Offs(pOrigin,170.10,23.91,0.00),v40,z0,tPen\WObj:=wPaper;
    MoveL Offs(pOrigin,193.26,21.58,0.00),v40,z0,tPen\WObj:=wPaper;
  ENDPROC

  PROC DrawPart5()
    MoveL Offs(pOrigin,193.69,20.94,0.00),v40,z0,tPen\WObj:=wPaper;
    MoveL Offs(pOrigin,193.19,19.73,0.00),v40,z0,tPen\WObj:=wPaper;
    MoveL Offs(pOrigin,191.35,19.66,0.00),v40,z0,tPen\WObj:=wPaper;
    MoveL Offs(pOrigin,157.99,23.27,0.00),v40,z0,tPen\WObj:=wPaper;
    MoveL Offs(pOrigin,157.99,23.27,0.00),v40,z0,tPen\WObj:=wPaper;
    MoveL Offs(pOrigin,156.93,23.27,0.00),v40,z0,tPen\WObj:=wPaper;
    MoveL Offs(pOrigin,156.29,23.91,0.00),v40,z0,tPen\WObj:=wPaper;
    MoveL Offs(pOrigin,156.29,23.91,0.00),v40,z0,tPen\WObj:=wPaper;
    MoveL Offs(pOrigin,156.50,24.55,0.00),v40,z0,tPen\WObj:=wPaper;
    MoveL Offs(pOrigin,156.93,24.55,0.00),v40,z0,tPen\WObj:=wPaper;
    MoveL Offs(pOrigin,156.29,24.55,0.00),v40,z0,tPen\WObj:=wPaper;
    MoveL Offs(pOrigin,155.65,25.19,0.00),v40,z0,tPen\WObj:=wPaper;
    MoveL Offs(pOrigin,154.80,25.12,0.00),v40,z0,tPen\WObj:=wPaper;
    MoveL Offs(pOrigin,153.52,24.12,0.00),v40,z0,tPen\WObj:=wPaper;
    MoveL Offs(pOrigin,150.76,24.34,0.00),v40,z0,tPen\WObj:=wPaper;
    MoveL Offs(pOrigin,149.70,24.76,0.00),v40,z0,tPen\WObj:=wPaper;
    MoveL Offs(pOrigin,149.70,24.76,0.00),v40,z0,tPen\WObj:=wPaper;
    MoveL Offs(pOrigin,147.79,24.76,0.00),v40,z0,tPen\WObj:=wPaper;
    MoveL Offs(pOrigin,147.57,25.19,0.00),v40,fine,tPen\WObj:=wPaper;
    MoveL Offs(pOrigin,147.57,25.19,6.00),v60,z5,tPen\WObj:=wPaper;
    MoveL Offs(pOrigin,147.44,26.77,6.00),vTravel,z5,tPen\WObj:=wPaper;
    MoveL Offs(pOrigin,147.44,26.77,0.00),v60,z0,tPen\WObj:=wPaper;
    MoveL Offs(pOrigin,141.43,20.76,0.00),v40,z0,tPen\WObj:=wPaper;
    MoveL Offs(pOrigin,141.33,20.20,0.00),v40,z0,tPen\WObj:=wPaper;
    MoveL Offs(pOrigin,132.77,28.77,0.00),v40,z0,tPen\WObj:=wPaper;
    MoveL Offs(pOrigin,132.47,28.22,0.00),v40,z0,tPen\WObj:=wPaper;
    MoveL Offs(pOrigin,129.16,24.92,0.00),v40,z0,tPen\WObj:=wPaper;
    MoveL Offs(pOrigin,128.41,24.17,0.00),v40,z0,tPen\WObj:=wPaper;
    MoveL Offs(pOrigin,126.61,22.36,0.00),v40,z0,tPen\WObj:=wPaper;
    MoveL Offs(pOrigin,126.50,21.60,0.00),v40,z0,tPen\WObj:=wPaper;
    MoveL Offs(pOrigin,117.93,30.16,0.00),v40,z0,tPen\WObj:=wPaper;
    MoveL Offs(pOrigin,117.34,29.53,0.00),v40,z0,tPen\WObj:=wPaper;
    MoveL Offs(pOrigin,111.78,23.97,0.00),v40,z0,tPen\WObj:=wPaper;
    MoveL Offs(pOrigin,111.51,23.14,0.00),v40,z0,tPen\WObj:=wPaper;
    MoveL Offs(pOrigin,103.10,31.56,0.00),v40,z0,tPen\WObj:=wPaper;
    MoveL Offs(pOrigin,102.52,31.13,0.00),v40,z0,tPen\WObj:=wPaper;
    MoveL Offs(pOrigin,96.81,25.42,0.00),v40,z0,tPen\WObj:=wPaper;
    MoveL Offs(pOrigin,96.79,25.56,0.00),v40,z0,tPen\WObj:=wPaper;
    MoveL Offs(pOrigin,109.75,25.56,0.00),v40,fine,tPen\WObj:=wPaper;
    MoveL Offs(pOrigin,109.75,25.56,6.00),v60,z5,tPen\WObj:=wPaper;
    MoveL Offs(pOrigin,110.29,23.96,6.00),vTravel,z5,tPen\WObj:=wPaper;
    MoveL Offs(pOrigin,110.29,23.96,0.00),v60,z0,tPen\WObj:=wPaper;
    MoveL Offs(pOrigin,116.15,29.82,0.00),v40,z0,tPen\WObj:=wPaper;
    MoveL Offs(pOrigin,116.44,30.17,0.00),v40,z0,tPen\WObj:=wPaper;
    MoveL Offs(pOrigin,124.70,21.90,0.00),v40,z0,tPen\WObj:=wPaper;
    MoveL Offs(pOrigin,125.11,22.36,0.00),v40,z0,tPen\WObj:=wPaper;
    MoveL Offs(pOrigin,126.91,24.16,0.00),v40,z0,tPen\WObj:=wPaper;
    MoveL Offs(pOrigin,127.67,24.91,0.00),v40,z0,tPen\WObj:=wPaper;
    MoveL Offs(pOrigin,130.97,28.22,0.00),v40,z0,tPen\WObj:=wPaper;
    MoveL Offs(pOrigin,130.97,29.07,0.00),v40,z0,tPen\WObj:=wPaper;
    MoveL Offs(pOrigin,139.54,20.51,0.00),v40,z0,tPen\WObj:=wPaper;
    MoveL Offs(pOrigin,140.09,20.91,0.00),v40,z0,tPen\WObj:=wPaper;
    MoveL Offs(pOrigin,141.89,22.71,0.00),v40,z0,tPen\WObj:=wPaper;
    MoveL Offs(pOrigin,142.64,23.46,0.00),v40,z0,tPen\WObj:=wPaper;
    MoveL Offs(pOrigin,146.10,26.92,0.00),v40,z0,tPen\WObj:=wPaper;
    MoveL Offs(pOrigin,145.95,27.53,0.00),v40,z0,tPen\WObj:=wPaper;
    MoveL Offs(pOrigin,154.82,18.66,0.00),v40,z0,tPen\WObj:=wPaper;
    MoveL Offs(pOrigin,155.06,19.45,0.00),v40,z0,tPen\WObj:=wPaper;
    MoveL Offs(pOrigin,158.97,23.36,0.00),v40,fine,tPen\WObj:=wPaper;
    MoveL Offs(pOrigin,158.97,23.36,6.00),v60,z5,tPen\WObj:=wPaper;
    MoveL Offs(pOrigin,157.77,23.66,6.00),vTravel,z5,tPen\WObj:=wPaper;
    MoveL Offs(pOrigin,157.77,23.66,0.00),v60,z0,tPen\WObj:=wPaper;
    MoveL Offs(pOrigin,153.71,19.60,0.00),v40,z0,tPen\WObj:=wPaper;
    MoveL Offs(pOrigin,153.02,18.97,0.00),v40,z0,tPen\WObj:=wPaper;
    MoveL Offs(pOrigin,144.31,27.68,0.00),v40,z0,tPen\WObj:=wPaper;
    MoveL Offs(pOrigin,144.75,27.06,0.00),v40,z0,tPen\WObj:=wPaper;
    MoveL Offs(pOrigin,143.70,26.01,0.00),v40,z0,tPen\WObj:=wPaper;
    MoveL Offs(pOrigin,142.95,25.26,0.00),v40,z0,tPen\WObj:=wPaper;
    MoveL Offs(pOrigin,141.44,23.76,0.00),v40,z0,tPen\WObj:=wPaper;
    MoveL Offs(pOrigin,141.41,24.50,0.00),v40,z0,tPen\WObj:=wPaper;
    MoveL Offs(pOrigin,139.07,24.50,0.00),v40,z0,tPen\WObj:=wPaper;
    MoveL Offs(pOrigin,138.60,23.90,0.00),v40,z0,tPen\WObj:=wPaper;
    MoveL Offs(pOrigin,141.90,27.20,0.00),v40,fine,tPen\WObj:=wPaper;
    MoveL Offs(pOrigin,141.90,27.20,6.00),v60,z5,tPen\WObj:=wPaper;
    MoveL Offs(pOrigin,140.56,25.83,6.00),vTravel,z5,tPen\WObj:=wPaper;
    MoveL Offs(pOrigin,140.56,25.83,0.00),v60,z0,tPen\WObj:=wPaper;
    MoveL Offs(pOrigin,141.20,25.05,0.00),v40,z0,tPen\WObj:=wPaper;
    MoveL Offs(pOrigin,142.48,24.76,0.00),v40,z0,tPen\WObj:=wPaper;
    MoveL Offs(pOrigin,143.96,24.76,0.00),v40,z0,tPen\WObj:=wPaper;
    MoveL Offs(pOrigin,144.60,25.40,0.00),v40,fine,tPen\WObj:=wPaper;
    MoveL Offs(pOrigin,144.60,25.40,6.00),v60,z5,tPen\WObj:=wPaper;
    MoveL Offs(pOrigin,147.75,27.22,6.00),vTravel,z5,tPen\WObj:=wPaper;
    MoveL Offs(pOrigin,147.75,27.22,0.00),v60,z0,tPen\WObj:=wPaper;
    MoveL Offs(pOrigin,156.47,18.51,0.00),v40,z0,tPen\WObj:=wPaper;
    MoveL Offs(pOrigin,156.41,19.31,0.00),v40,z0,tPen\WObj:=wPaper;
    MoveL Offs(pOrigin,158.21,21.11,0.00),v40,z0,tPen\WObj:=wPaper;
    MoveL Offs(pOrigin,158.96,21.86,0.00),v40,z0,tPen\WObj:=wPaper;
    MoveL Offs(pOrigin,160.47,23.37,0.00),v40,z0,tPen\WObj:=wPaper;
    MoveL Offs(pOrigin,159.90,22.39,0.00),v40,z0,tPen\WObj:=wPaper;
    MoveL Offs(pOrigin,162.66,22.39,0.00),v40,z0,tPen\WObj:=wPaper;
    MoveL Offs(pOrigin,163.16,23.07,0.00),v40,z0,tPen\WObj:=wPaper;
    MoveL Offs(pOrigin,158.95,18.87,0.00),v40,fine,tPen\WObj:=wPaper;
    MoveL Offs(pOrigin,158.95,18.87,6.00),v60,z5,tPen\WObj:=wPaper;
    MoveL Offs(pOrigin,157.76,19.16,6.00),vTravel,z5,tPen\WObj:=wPaper;
    MoveL Offs(pOrigin,157.76,19.16,0.00),v60,z0,tPen\WObj:=wPaper;
    MoveL Offs(pOrigin,161.81,23.22,0.00),v40,fine,tPen\WObj:=wPaper;
    MoveL Offs(pOrigin,161.81,23.22,6.00),v60,z5,tPen\WObj:=wPaper;
    MoveL Offs(pOrigin,161.52,24.42,6.00),vTravel,z5,tPen\WObj:=wPaper;
    MoveL Offs(pOrigin,161.52,24.42,0.00),v60,z0,tPen\WObj:=wPaper;
    MoveL Offs(pOrigin,162.72,25.62,0.00),v40,z0,tPen\WObj:=wPaper;
    MoveL Offs(pOrigin,162.44,25.98,0.00),v40,z0,tPen\WObj:=wPaper;
    MoveL Offs(pOrigin,171.45,16.97,0.00),v40,fine,tPen\WObj:=wPaper;
    MoveL Offs(pOrigin,171.45,16.97,6.00),v60,z5,tPen\WObj:=wPaper;
    MoveL Offs(pOrigin,172.58,17.56,6.00),vTravel,z5,tPen\WObj:=wPaper;
    MoveL Offs(pOrigin,172.58,17.56,0.00),v60,z0,tPen\WObj:=wPaper;
    MoveL Offs(pOrigin,176.64,21.62,0.00),v40,fine,tPen\WObj:=wPaper;
    MoveL Offs(pOrigin,176.64,21.62,6.00),v60,z5,tPen\WObj:=wPaper;
    MoveL Offs(pOrigin,177.99,21.47,6.00),vTravel,z5,tPen\WObj:=wPaper;
    MoveL Offs(pOrigin,177.99,21.47,0.00),v60,z0,tPen\WObj:=wPaper;
    MoveL Offs(pOrigin,173.78,17.26,0.00),v40,z0,tPen\WObj:=wPaper;
    MoveL Offs(pOrigin,173.10,16.81,0.00),v40,z0,tPen\WObj:=wPaper;
    MoveL Offs(pOrigin,164.24,25.68,0.00),v40,z0,tPen\WObj:=wPaper;
    MoveL Offs(pOrigin,163.92,25.32,0.00),v40,z0,tPen\WObj:=wPaper;
    MoveL Offs(pOrigin,163.02,24.42,0.00),v40,fine,tPen\WObj:=wPaper;
    MoveL Offs(pOrigin,163.02,24.42,6.00),v60,z5,tPen\WObj:=wPaper;
    MoveL Offs(pOrigin,164.36,24.28,6.00),vTravel,z5,tPen\WObj:=wPaper;
    MoveL Offs(pOrigin,164.36,24.28,0.00),v60,z0,tPen\WObj:=wPaper;
    MoveL Offs(pOrigin,165.27,25.18,0.00),v40,z0,tPen\WObj:=wPaper;
    MoveL Offs(pOrigin,165.73,25.67,0.00),v40,z0,tPen\WObj:=wPaper;
    MoveL Offs(pOrigin,174.90,16.51,0.00),v40,z0,tPen\WObj:=wPaper;
  ENDPROC

  PROC DrawPart6()
    MoveL Offs(pOrigin,175.13,17.12,0.00),v40,z0,tPen\WObj:=wPaper;
    MoveL Offs(pOrigin,179.18,21.18,0.00),v40,fine,tPen\WObj:=wPaper;
    MoveL Offs(pOrigin,179.18,21.18,6.00),v60,z5,tPen\WObj:=wPaper;
    MoveL Offs(pOrigin,178.18,20.28,6.00),vTravel,z5,tPen\WObj:=wPaper;
    MoveL Offs(pOrigin,178.18,20.28,0.00),v60,z0,tPen\WObj:=wPaper;
    MoveL Offs(pOrigin,183.91,20.28,0.00),v40,z0,tPen\WObj:=wPaper;
    MoveL Offs(pOrigin,183.53,21.04,0.00),v40,z0,tPen\WObj:=wPaper;
    MoveL Offs(pOrigin,179.17,16.68,0.00),v40,z0,tPen\WObj:=wPaper;
    MoveL Offs(pOrigin,178.81,17.11,0.00),v40,z0,tPen\WObj:=wPaper;
    MoveL Offs(pOrigin,195.18,17.11,0.00),v40,z0,tPen\WObj:=wPaper;
    MoveL Offs(pOrigin,196.10,17.18,0.00),v40,z0,tPen\WObj:=wPaper;
    MoveL Offs(pOrigin,193.70,14.78,0.00),v40,z0,tPen\WObj:=wPaper;
    MoveL Offs(pOrigin,193.90,15.00,0.00),v40,z0,tPen\WObj:=wPaper;
    MoveL Offs(pOrigin,202.82,15.00,0.00),v40,z0,tPen\WObj:=wPaper;
    MoveL Offs(pOrigin,203.43,15.56,0.00),v40,z0,tPen\WObj:=wPaper;
    MoveL Offs(pOrigin,201.48,13.60,0.00),v40,z0,tPen\WObj:=wPaper;
    MoveL Offs(pOrigin,200.83,12.98,0.00),v40,z0,tPen\WObj:=wPaper;
    MoveL Offs(pOrigin,190.31,23.50,0.00),v40,z0,tPen\WObj:=wPaper;
    MoveL Offs(pOrigin,189.98,23.01,0.00),v40,z0,tPen\WObj:=wPaper;
    MoveL Offs(pOrigin,188.77,21.80,0.00),v40,fine,tPen\WObj:=wPaper;
    MoveL Offs(pOrigin,188.77,21.80,6.00),v60,z5,tPen\WObj:=wPaper;
    MoveL Offs(pOrigin,187.58,22.10,6.00),vTravel,z5,tPen\WObj:=wPaper;
    MoveL Offs(pOrigin,187.58,22.10,0.00),v60,z0,tPen\WObj:=wPaper;
    MoveL Offs(pOrigin,188.63,23.15,0.00),v40,z0,tPen\WObj:=wPaper;
    MoveL Offs(pOrigin,188.66,23.65,0.00),v40,z0,tPen\WObj:=wPaper;
    MoveL Offs(pOrigin,199.03,13.29,0.00),v40,z0,tPen\WObj:=wPaper;
    MoveL Offs(pOrigin,198.64,13.75,0.00),v40,z0,tPen\WObj:=wPaper;
    MoveL Offs(pOrigin,200.89,16.00,0.00),v40,z0,tPen\WObj:=wPaper;
    MoveL Offs(pOrigin,201.86,16.42,0.00),v40,z0,tPen\WObj:=wPaper;
    MoveL Offs(pOrigin,205.77,12.52,0.00),v40,z0,tPen\WObj:=wPaper;
    MoveL Offs(pOrigin,205.52,13.17,0.00),v40,z0,tPen\WObj:=wPaper;
    MoveL Offs(pOrigin,210.78,18.43,0.00),v40,z0,tPen\WObj:=wPaper;
    MoveL Offs(pOrigin,210.05,18.17,0.00),v40,z0,tPen\WObj:=wPaper;
    MoveL Offs(pOrigin,206.44,18.17,0.00),v40,z0,tPen\WObj:=wPaper;
    MoveL Offs(pOrigin,205.84,17.96,0.00),v40,z0,tPen\WObj:=wPaper;
    MoveL Offs(pOrigin,210.50,22.62,0.00),v40,z0,tPen\WObj:=wPaper;
    MoveL Offs(pOrigin,210.23,22.99,0.00),v40,z0,tPen\WObj:=wPaper;
    MoveL Offs(pOrigin,221.50,11.72,0.00),v40,z0,tPen\WObj:=wPaper;
    MoveL Offs(pOrigin,221.25,12.47,0.00),v40,z0,tPen\WObj:=wPaper;
    MoveL Offs(pOrigin,225.16,16.37,0.00),v40,fine,tPen\WObj:=wPaper;
    MoveL Offs(pOrigin,225.16,16.37,6.00),v60,z5,tPen\WObj:=wPaper;
    MoveL Offs(pOrigin,225.01,17.72,6.00),vTravel,z5,tPen\WObj:=wPaper;
    MoveL Offs(pOrigin,225.01,17.72,0.00),v60,z0,tPen\WObj:=wPaper;
    MoveL Offs(pOrigin,226.67,19.37,0.00),v40,z0,tPen\WObj:=wPaper;
    MoveL Offs(pOrigin,226.87,19.79,0.00),v40,z0,tPen\WObj:=wPaper;
    MoveL Offs(pOrigin,235.89,10.78,0.00),v40,z0,tPen\WObj:=wPaper;
    MoveL Offs(pOrigin,235.18,11.46,0.00),v40,z0,tPen\WObj:=wPaper;
    MoveL Offs(pOrigin,238.34,14.62,0.00),v40,z0,tPen\WObj:=wPaper;
    MoveL Offs(pOrigin,238.95,13.94,0.00),v40,z0,tPen\WObj:=wPaper;
    MoveL Offs(pOrigin,244.69,13.94,0.00),v40,z0,tPen\WObj:=wPaper;
    MoveL Offs(pOrigin,245.22,14.04,0.00),v40,z0,tPen\WObj:=wPaper;
    MoveL Offs(pOrigin,248.38,17.19,0.00),v40,z0,tPen\WObj:=wPaper;
    MoveL Offs(pOrigin,247.78,18.09,0.00),v40,z0,tPen\WObj:=wPaper;
    MoveL Offs(pOrigin,253.34,23.65,0.00),v40,z0,tPen\WObj:=wPaper;
    MoveL Offs(pOrigin,253.97,24.05,0.00),v40,z0,tPen\WObj:=wPaper;
    MoveL Offs(pOrigin,260.58,17.44,0.00),v40,z0,tPen\WObj:=wPaper;
    MoveL Offs(pOrigin,261.27,18.13,0.00),v40,z0,tPen\WObj:=wPaper;
    MoveL Offs(pOrigin,264.57,21.44,0.00),v40,z0,tPen\WObj:=wPaper;
    MoveL Offs(pOrigin,263.97,22.34,0.00),v40,z0,tPen\WObj:=wPaper;
    MoveL Offs(pOrigin,272.99,31.35,0.00),v40,z0,tPen\WObj:=wPaper;
    MoveL Offs(pOrigin,273.12,31.78,0.00),v40,z0,tPen\WObj:=wPaper;
    MoveL Offs(pOrigin,275.68,29.23,0.00),v40,z0,tPen\WObj:=wPaper;
    MoveL Offs(pOrigin,275.08,28.96,0.00),v40,z0,tPen\WObj:=wPaper;
    MoveL Offs(pOrigin,269.97,23.85,0.00),v40,z0,tPen\WObj:=wPaper;
    MoveL Offs(pOrigin,270.83,24.34,0.00),v40,z0,tPen\WObj:=wPaper;
    MoveL Offs(pOrigin,269.34,23.91,0.00),v40,z0,tPen\WObj:=wPaper;
    MoveL Offs(pOrigin,269.12,24.55,0.00),v40,z0,tPen\WObj:=wPaper;
    MoveL Offs(pOrigin,269.12,24.55,0.00),v40,z0,tPen\WObj:=wPaper;
    MoveL Offs(pOrigin,270.83,24.98,0.00),v40,fine,tPen\WObj:=wPaper;
    MoveL Offs(pOrigin,270.83,24.98,6.00),v60,z5,tPen\WObj:=wPaper;
    MoveL Offs(pOrigin,272.22,24.61,6.00),vTravel,z5,tPen\WObj:=wPaper;
    MoveL Offs(pOrigin,272.22,24.61,0.00),v60,z0,tPen\WObj:=wPaper;
    MoveL Offs(pOrigin,275.23,27.61,0.00),v40,z0,tPen\WObj:=wPaper;
    MoveL Offs(pOrigin,274.86,27.67,0.00),v40,z0,tPen\WObj:=wPaper;
    MoveL Offs(pOrigin,270.82,27.67,0.00),v40,z0,tPen\WObj:=wPaper;
    MoveL Offs(pOrigin,270.40,26.62,0.00),v40,z0,tPen\WObj:=wPaper;
    MoveL Offs(pOrigin,268.27,26.62,0.00),v40,fine,tPen\WObj:=wPaper;
    MoveL Offs(pOrigin,268.27,26.62,6.00),v60,z5,tPen\WObj:=wPaper;
    MoveL Offs(pOrigin,266.36,25.56,6.00),vTravel,z5,tPen\WObj:=wPaper;
    MoveL Offs(pOrigin,266.36,25.56,0.00),v60,z0,tPen\WObj:=wPaper;
    MoveL Offs(pOrigin,264.02,25.56,0.00),v40,z0,tPen\WObj:=wPaper;
    MoveL Offs(pOrigin,263.39,26.23,0.00),v40,z0,tPen\WObj:=wPaper;
    MoveL Offs(pOrigin,257.98,20.82,0.00),v40,z0,tPen\WObj:=wPaper;
    MoveL Offs(pOrigin,257.65,20.94,0.00),v40,z0,tPen\WObj:=wPaper;
    MoveL Offs(pOrigin,259.35,21.36,0.00),v40,z0,tPen\WObj:=wPaper;
    MoveL Offs(pOrigin,259.35,22.00,0.00),v40,z0,tPen\WObj:=wPaper;
    MoveL Offs(pOrigin,259.56,21.36,0.00),v40,z0,tPen\WObj:=wPaper;
    MoveL Offs(pOrigin,260.20,21.58,0.00),v40,z0,tPen\WObj:=wPaper;
    MoveL Offs(pOrigin,260.20,21.58,0.00),v40,z0,tPen\WObj:=wPaper;
    MoveL Offs(pOrigin,264.24,22.64,0.00),v40,z0,tPen\WObj:=wPaper;
    MoveL Offs(pOrigin,264.24,23.27,0.00),v40,z0,tPen\WObj:=wPaper;
    MoveL Offs(pOrigin,260.20,22.21,0.00),v40,z0,tPen\WObj:=wPaper;
    MoveL Offs(pOrigin,260.08,21.42,0.00),v40,z0,tPen\WObj:=wPaper;
    MoveL Offs(pOrigin,268.94,30.29,0.00),v40,z0,tPen\WObj:=wPaper;
    MoveL Offs(pOrigin,268.33,30.60,0.00),v40,z0,tPen\WObj:=wPaper;
    MoveL Offs(pOrigin,277.20,21.73,0.00),v40,z0,tPen\WObj:=wPaper;
    MoveL Offs(pOrigin,277.46,22.38,0.00),v40,z0,tPen\WObj:=wPaper;
    MoveL Offs(pOrigin,279.56,24.48,0.00),v40,z0,tPen\WObj:=wPaper;
    MoveL Offs(pOrigin,279.88,25.02,0.00),v40,z0,tPen\WObj:=wPaper;
    MoveL Offs(pOrigin,282.89,22.02,0.00),v40,z0,tPen\WObj:=wPaper;
    MoveL Offs(pOrigin,281.95,22.39,0.00),v40,z0,tPen\WObj:=wPaper;
    MoveL Offs(pOrigin,284.20,24.64,0.00),v40,z0,tPen\WObj:=wPaper;
    MoveL Offs(pOrigin,284.23,25.16,0.00),v40,z0,tPen\WObj:=wPaper;
    MoveL Offs(pOrigin,286.78,22.60,0.00),v40,z0,tPen\WObj:=wPaper;
    MoveL Offs(pOrigin,286.76,23.45,0.00),v40,z0,tPen\WObj:=wPaper;
    MoveL Offs(pOrigin,274.65,23.45,0.00),v40,z0,tPen\WObj:=wPaper;
    MoveL Offs(pOrigin,275.63,23.06,0.00),v40,z0,tPen\WObj:=wPaper;
    MoveL Offs(pOrigin,275.63,25.40,0.00),v40,z0,tPen\WObj:=wPaper;
    MoveL Offs(pOrigin,276.14,25.56,0.00),v40,z0,tPen\WObj:=wPaper;
    MoveL Offs(pOrigin,273.59,25.56,0.00),v40,z0,tPen\WObj:=wPaper;
    MoveL Offs(pOrigin,273.38,25.61,0.00),v40,z0,tPen\WObj:=wPaper;
    MoveL Offs(pOrigin,274.01,26.04,0.00),v40,z0,tPen\WObj:=wPaper;
    MoveL Offs(pOrigin,273.80,26.89,0.00),v40,z0,tPen\WObj:=wPaper;
    MoveL Offs(pOrigin,273.16,27.10,0.00),v40,z0,tPen\WObj:=wPaper;
    MoveL Offs(pOrigin,234.06,17.33,0.00),v40,z0,tPen\WObj:=wPaper;
    MoveL Offs(pOrigin,212.39,19.45,0.00),v40,z0,tPen\WObj:=wPaper;
    MoveL Offs(pOrigin,210.26,19.38,0.00),v40,z0,tPen\WObj:=wPaper;
    MoveL Offs(pOrigin,209.70,17.96,0.00),v40,z0,tPen\WObj:=wPaper;
    MoveL Offs(pOrigin,210.26,17.54,0.00),v40,z0,tPen\WObj:=wPaper;
    MoveL Offs(pOrigin,233.64,15.41,0.00),v40,z0,tPen\WObj:=wPaper;
  ENDPROC

  PROC DrawPart7()
    MoveL Offs(pOrigin,250.43,19.66,0.00),v40,z0,tPen\WObj:=wPaper;
    MoveL Offs(pOrigin,250.43,19.02,0.00),v40,z0,tPen\WObj:=wPaper;
    MoveL Offs(pOrigin,233.64,14.56,0.00),v40,z0,tPen\WObj:=wPaper;
    MoveL Offs(pOrigin,230.45,14.56,0.00),v40,z0,tPen\WObj:=wPaper;
    MoveL Offs(pOrigin,212.39,16.48,0.00),v40,z0,tPen\WObj:=wPaper;
    MoveL Offs(pOrigin,210.05,16.48,0.00),v40,z0,tPen\WObj:=wPaper;
    MoveL Offs(pOrigin,209.62,15.84,0.00),v40,z0,tPen\WObj:=wPaper;
    MoveL Offs(pOrigin,210.26,15.20,0.00),v40,z0,tPen\WObj:=wPaper;
    MoveL Offs(pOrigin,230.45,13.07,0.00),v40,z0,tPen\WObj:=wPaper;
    MoveL Offs(pOrigin,234.91,13.07,0.00),v40,z0,tPen\WObj:=wPaper;
    MoveL Offs(pOrigin,274.01,23.27,0.00),v40,z0,tPen\WObj:=wPaper;
    MoveL Offs(pOrigin,275.29,23.91,0.00),v40,z0,tPen\WObj:=wPaper;
    MoveL Offs(pOrigin,274.86,25.12,0.00),v40,z0,tPen\WObj:=wPaper;
    MoveL Offs(pOrigin,273.38,24.98,0.00),v40,z0,tPen\WObj:=wPaper;
    MoveL Offs(pOrigin,273.38,24.98,0.00),v40,z0,tPen\WObj:=wPaper;
    MoveL Offs(pOrigin,272.74,24.76,0.00),v40,z0,tPen\WObj:=wPaper;
    MoveL Offs(pOrigin,272.52,25.40,0.00),v40,fine,tPen\WObj:=wPaper;
    MoveL Offs(pOrigin,272.52,25.40,6.00),v60,z5,tPen\WObj:=wPaper;
    MoveL Offs(pOrigin,273.16,26.62,6.00),vTravel,z5,tPen\WObj:=wPaper;
    MoveL Offs(pOrigin,273.16,26.62,0.00),v60,z0,tPen\WObj:=wPaper;
    MoveL Offs(pOrigin,275.50,26.62,0.00),v40,z0,tPen\WObj:=wPaper;
    MoveL Offs(pOrigin,275.50,26.46,0.00),v40,z0,tPen\WObj:=wPaper;
    MoveL Offs(pOrigin,275.29,26.89,0.00),v40,z0,tPen\WObj:=wPaper;
    MoveL Offs(pOrigin,275.50,26.46,0.00),v40,z0,tPen\WObj:=wPaper;
    MoveL Offs(pOrigin,275.82,26.72,0.00),v40,z0,tPen\WObj:=wPaper;
    MoveL Offs(pOrigin,273.72,24.61,0.00),v40,z0,tPen\WObj:=wPaper;
    MoveL Offs(pOrigin,274.86,24.50,0.00),v40,z0,tPen\WObj:=wPaper;
    MoveL Offs(pOrigin,277.84,24.50,0.00),v40,z0,tPen\WObj:=wPaper;
    MoveL Offs(pOrigin,278.21,24.63,0.00),v40,z0,tPen\WObj:=wPaper;
    MoveL Offs(pOrigin,275.81,22.22,0.00),v40,z0,tPen\WObj:=wPaper;
    MoveL Offs(pOrigin,275.71,22.39,0.00),v40,z0,tPen\WObj:=wPaper;
    MoveL Offs(pOrigin,270.82,22.39,0.00),v40,z0,tPen\WObj:=wPaper;
    MoveL Offs(pOrigin,270.57,22.95,0.00),v40,z0,tPen\WObj:=wPaper;
    MoveL Offs(pOrigin,267.41,19.80,0.00),v40,z0,tPen\WObj:=wPaper;
    MoveL Offs(pOrigin,267.62,19.37,0.00),v40,z0,tPen\WObj:=wPaper;
    MoveL Offs(pOrigin,253.49,33.49,0.00),v40,z0,tPen\WObj:=wPaper;
    MoveL Offs(pOrigin,254.39,34.09,0.00),v40,z0,tPen\WObj:=wPaper;
    MoveL Offs(pOrigin,256.49,31.98,0.00),v40,z0,tPen\WObj:=wPaper;
    MoveL Offs(pOrigin,255.52,31.90,0.00),v40,z0,tPen\WObj:=wPaper;
    MoveL Offs(pOrigin,252.76,31.90,0.00),v40,z0,tPen\WObj:=wPaper;
    MoveL Offs(pOrigin,252.40,31.35,0.00),v40,z0,tPen\WObj:=wPaper;
    MoveL Offs(pOrigin,252.40,30.08,0.00),v40,z0,tPen\WObj:=wPaper;
    MoveL Offs(pOrigin,251.91,30.08,0.00),v40,z0,tPen\WObj:=wPaper;
    MoveL Offs(pOrigin,252.12,29.30,0.00),v40,z0,tPen\WObj:=wPaper;
    MoveL Offs(pOrigin,254.46,29.51,0.00),v40,z0,tPen\WObj:=wPaper;
    MoveL Offs(pOrigin,256.16,28.30,0.00),v40,z0,tPen\WObj:=wPaper;
    MoveL Offs(pOrigin,258.08,27.74,0.00),v40,z0,tPen\WObj:=wPaper;
    MoveL Offs(pOrigin,264.88,27.74,0.00),v40,z0,tPen\WObj:=wPaper;
    MoveL Offs(pOrigin,269.12,28.59,0.00),v40,z0,tPen\WObj:=wPaper;
    MoveL Offs(pOrigin,272.10,28.59,0.00),v40,z0,tPen\WObj:=wPaper;
    MoveL Offs(pOrigin,272.10,28.59,0.00),v40,z0,tPen\WObj:=wPaper;
    MoveL Offs(pOrigin,271.67,27.81,0.00),v40,z0,tPen\WObj:=wPaper;
    MoveL Offs(pOrigin,233.64,18.39,0.00),v40,z0,tPen\WObj:=wPaper;
    MoveL Offs(pOrigin,214.94,20.09,0.00),v40,z0,tPen\WObj:=wPaper;
    MoveL Offs(pOrigin,214.09,20.51,0.00),v40,z0,tPen\WObj:=wPaper;
    MoveL Offs(pOrigin,214.09,20.51,0.00),v40,z0,tPen\WObj:=wPaper;
    MoveL Offs(pOrigin,214.51,21.08,0.00),v40,z0,tPen\WObj:=wPaper;
    MoveL Offs(pOrigin,245.75,27.95,0.00),v40,z0,tPen\WObj:=wPaper;
    MoveL Offs(pOrigin,245.57,27.82,0.00),v40,z0,tPen\WObj:=wPaper;
    MoveL Offs(pOrigin,249.62,31.88,0.00),v40,z0,tPen\WObj:=wPaper;
    MoveL Offs(pOrigin,250.00,31.56,0.00),v40,z0,tPen\WObj:=wPaper;
    MoveL Offs(pOrigin,251.35,33.69,0.00),v40,z0,tPen\WObj:=wPaper;
    MoveL Offs(pOrigin,251.49,34.75,0.00),v40,z0,tPen\WObj:=wPaper;
    MoveL Offs(pOrigin,250.43,36.88,0.00),v40,z0,tPen\WObj:=wPaper;
    MoveL Offs(pOrigin,249.57,37.65,0.00),v40,z0,tPen\WObj:=wPaper;
    MoveL Offs(pOrigin,248.51,37.94,0.00),v40,z0,tPen\WObj:=wPaper;
    MoveL Offs(pOrigin,248.30,38.23,0.00),v40,z0,tPen\WObj:=wPaper;
    MoveL Offs(pOrigin,246.60,38.23,0.00),v40,z0,tPen\WObj:=wPaper;
    MoveL Offs(pOrigin,247.02,38.79,0.00),v40,z0,tPen\WObj:=wPaper;
    MoveL Offs(pOrigin,247.66,39.42,0.00),v40,z0,tPen\WObj:=wPaper;
    MoveL Offs(pOrigin,247.02,38.79,0.00),v40,z0,tPen\WObj:=wPaper;
    MoveL Offs(pOrigin,247.66,39.29,0.00),v40,z0,tPen\WObj:=wPaper;
    MoveL Offs(pOrigin,249.15,39.29,0.00),v40,z0,tPen\WObj:=wPaper;
    MoveL Offs(pOrigin,249.88,38.60,0.00),v40,z0,tPen\WObj:=wPaper;
    MoveL Offs(pOrigin,244.02,44.46,0.00),v40,z0,tPen\WObj:=wPaper;
    MoveL Offs(pOrigin,244.62,45.35,0.00),v40,z0,tPen\WObj:=wPaper;
    MoveL Offs(pOrigin,246.87,43.10,0.00),v40,z0,tPen\WObj:=wPaper;
    MoveL Offs(pOrigin,246.18,43.51,0.00),v40,z0,tPen\WObj:=wPaper;
    MoveL Offs(pOrigin,244.69,43.51,0.00),v40,z0,tPen\WObj:=wPaper;
    MoveL Offs(pOrigin,244.05,43.25,0.00),v40,z0,tPen\WObj:=wPaper;
    MoveL Offs(pOrigin,244.48,43.67,0.00),v40,z0,tPen\WObj:=wPaper;
    MoveL Offs(pOrigin,244.05,43.25,0.00),v40,z0,tPen\WObj:=wPaper;
    MoveL Offs(pOrigin,243.42,43.56,0.00),v40,z0,tPen\WObj:=wPaper;
    MoveL Offs(pOrigin,249.59,37.40,0.00),v40,z0,tPen\WObj:=wPaper;
    MoveL Offs(pOrigin,248.54,36.95,0.00),v40,z0,tPen\WObj:=wPaper;
    MoveL Offs(pOrigin,246.13,39.36,0.00),v40,z0,tPen\WObj:=wPaper;
    MoveL Offs(pOrigin,245.39,38.61,0.00),v40,z0,tPen\WObj:=wPaper;
    MoveL Offs(pOrigin,247.64,36.36,0.00),v40,z0,tPen\WObj:=wPaper;
    MoveL Offs(pOrigin,247.02,37.18,0.00),v40,z0,tPen\WObj:=wPaper;
    MoveL Offs(pOrigin,245.54,37.18,0.00),v40,z0,tPen\WObj:=wPaper;
    MoveL Offs(pOrigin,245.96,36.12,0.00),v40,z0,tPen\WObj:=wPaper;
    MoveL Offs(pOrigin,244.48,36.12,0.00),v40,z0,tPen\WObj:=wPaper;
    MoveL Offs(pOrigin,244.69,36.24,0.00),v40,z0,tPen\WObj:=wPaper;
    MoveL Offs(pOrigin,244.90,36.66,0.00),v40,z0,tPen\WObj:=wPaper;
    MoveL Offs(pOrigin,244.69,36.24,0.00),v40,z0,tPen\WObj:=wPaper;
    MoveL Offs(pOrigin,244.10,36.80,0.00),v40,z0,tPen\WObj:=wPaper;
    MoveL Offs(pOrigin,241.99,34.70,0.00),v40,z0,tPen\WObj:=wPaper;
    MoveL Offs(pOrigin,242.35,35.06,0.00),v40,z0,tPen\WObj:=wPaper;
    MoveL Offs(pOrigin,245.54,35.06,0.00),v40,z0,tPen\WObj:=wPaper;
    MoveL Offs(pOrigin,246.30,34.71,0.00),v40,z0,tPen\WObj:=wPaper;
    MoveL Offs(pOrigin,237.73,43.28,0.00),v40,fine,tPen\WObj:=wPaper;
    MoveL Offs(pOrigin,237.73,43.28,6.00),v60,z5,tPen\WObj:=wPaper;
    MoveL Offs(pOrigin,238.03,44.47,6.00),vTravel,z5,tPen\WObj:=wPaper;
    MoveL Offs(pOrigin,238.03,44.47,0.00),v60,z0,tPen\WObj:=wPaper;
    MoveL Offs(pOrigin,239.68,42.82,0.00),v40,fine,tPen\WObj:=wPaper;
    MoveL Offs(pOrigin,239.68,42.82,6.00),v60,z5,tPen\WObj:=wPaper;
    MoveL Offs(pOrigin,239.68,44.32,6.00),vTravel,z5,tPen\WObj:=wPaper;
    MoveL Offs(pOrigin,239.68,44.32,0.00),v60,z0,tPen\WObj:=wPaper;
    MoveL Offs(pOrigin,238.02,45.97,0.00),v40,fine,tPen\WObj:=wPaper;
    MoveL Offs(pOrigin,238.02,45.97,6.00),v60,z5,tPen\WObj:=wPaper;
    MoveL Offs(pOrigin,238.02,47.47,6.00),vTravel,z5,tPen\WObj:=wPaper;
    MoveL Offs(pOrigin,238.02,47.47,0.00),v60,z0,tPen\WObj:=wPaper;
    MoveL Offs(pOrigin,239.97,45.52,0.00),v40,fine,tPen\WObj:=wPaper;
    MoveL Offs(pOrigin,239.97,45.52,6.00),v60,z5,tPen\WObj:=wPaper;
    MoveL Offs(pOrigin,239.97,47.01,6.00),vTravel,z5,tPen\WObj:=wPaper;
    MoveL Offs(pOrigin,239.97,47.01,0.00),v60,z0,tPen\WObj:=wPaper;
    MoveL Offs(pOrigin,238.17,48.82,0.00),v40,fine,tPen\WObj:=wPaper;
    MoveL Offs(pOrigin,238.17,48.82,6.00),v60,z5,tPen\WObj:=wPaper;
    MoveL Offs(pOrigin,238.16,50.32,6.00),vTravel,z5,tPen\WObj:=wPaper;
    MoveL Offs(pOrigin,238.16,50.32,0.00),v60,z0,tPen\WObj:=wPaper;
  ENDPROC

  PROC DrawPart8()
    MoveL Offs(pOrigin,240.11,48.36,0.00),v40,fine,tPen\WObj:=wPaper;
    MoveL Offs(pOrigin,240.11,48.36,6.00),v60,z5,tPen\WObj:=wPaper;
    MoveL Offs(pOrigin,240.11,49.86,6.00),vTravel,z5,tPen\WObj:=wPaper;
    MoveL Offs(pOrigin,240.11,49.86,0.00),v60,z0,tPen\WObj:=wPaper;
    MoveL Offs(pOrigin,238.31,51.66,0.00),v40,fine,tPen\WObj:=wPaper;
    MoveL Offs(pOrigin,238.31,51.66,6.00),v60,z5,tPen\WObj:=wPaper;
    MoveL Offs(pOrigin,238.30,53.16,6.00),vTravel,z5,tPen\WObj:=wPaper;
    MoveL Offs(pOrigin,238.30,53.16,0.00),v60,z0,tPen\WObj:=wPaper;
    MoveL Offs(pOrigin,240.41,51.06,0.00),v40,fine,tPen\WObj:=wPaper;
    MoveL Offs(pOrigin,240.41,51.06,6.00),v60,z5,tPen\WObj:=wPaper;
    MoveL Offs(pOrigin,240.55,52.41,6.00),vTravel,z5,tPen\WObj:=wPaper;
    MoveL Offs(pOrigin,240.55,52.41,0.00),v60,z0,tPen\WObj:=wPaper;
    MoveL Offs(pOrigin,238.60,54.36,0.00),v40,fine,tPen\WObj:=wPaper;
    MoveL Offs(pOrigin,238.60,54.36,6.00),v60,z5,tPen\WObj:=wPaper;
    MoveL Offs(pOrigin,238.74,55.71,6.00),vTravel,z5,tPen\WObj:=wPaper;
    MoveL Offs(pOrigin,238.74,55.71,0.00),v60,z0,tPen\WObj:=wPaper;
    MoveL Offs(pOrigin,240.55,53.90,0.00),v40,fine,tPen\WObj:=wPaper;
    MoveL Offs(pOrigin,240.55,53.90,6.00),v60,z5,tPen\WObj:=wPaper;
    MoveL Offs(pOrigin,240.69,55.25,6.00),vTravel,z5,tPen\WObj:=wPaper;
    MoveL Offs(pOrigin,240.69,55.25,0.00),v60,z0,tPen\WObj:=wPaper;
    MoveL Offs(pOrigin,238.74,57.20,0.00),v40,fine,tPen\WObj:=wPaper;
    MoveL Offs(pOrigin,238.74,57.20,6.00),v60,z5,tPen\WObj:=wPaper;
    MoveL Offs(pOrigin,239.04,58.40,6.00),vTravel,z5,tPen\WObj:=wPaper;
    MoveL Offs(pOrigin,239.04,58.40,0.00),v60,z0,tPen\WObj:=wPaper;
    MoveL Offs(pOrigin,240.99,56.45,0.00),v40,fine,tPen\WObj:=wPaper;
    MoveL Offs(pOrigin,240.99,56.45,6.00),v60,z5,tPen\WObj:=wPaper;
    MoveL Offs(pOrigin,241.13,57.80,6.00),vTravel,z5,tPen\WObj:=wPaper;
    MoveL Offs(pOrigin,241.13,57.80,0.00),v60,z0,tPen\WObj:=wPaper;
    MoveL Offs(pOrigin,239.18,59.75,0.00),v40,fine,tPen\WObj:=wPaper;
    MoveL Offs(pOrigin,239.18,59.75,6.00),v60,z5,tPen\WObj:=wPaper;
    MoveL Offs(pOrigin,239.33,61.10,6.00),vTravel,z5,tPen\WObj:=wPaper;
    MoveL Offs(pOrigin,239.33,61.10,0.00),v60,z0,tPen\WObj:=wPaper;
    MoveL Offs(pOrigin,241.28,59.14,0.00),v40,fine,tPen\WObj:=wPaper;
    MoveL Offs(pOrigin,241.28,59.14,6.00),v60,z5,tPen\WObj:=wPaper;
    MoveL Offs(pOrigin,241.28,60.64,6.00),vTravel,z5,tPen\WObj:=wPaper;
    MoveL Offs(pOrigin,241.28,60.64,0.00),v60,z0,tPen\WObj:=wPaper;
    MoveL Offs(pOrigin,239.47,62.45,0.00),v40,fine,tPen\WObj:=wPaper;
    MoveL Offs(pOrigin,239.47,62.45,6.00),v60,z5,tPen\WObj:=wPaper;
    MoveL Offs(pOrigin,239.47,63.94,6.00),vTravel,z5,tPen\WObj:=wPaper;
    MoveL Offs(pOrigin,239.47,63.94,0.00),v60,z0,tPen\WObj:=wPaper;
    MoveL Offs(pOrigin,241.57,61.84,0.00),v40,fine,tPen\WObj:=wPaper;
    MoveL Offs(pOrigin,241.57,61.84,6.00),v60,z5,tPen\WObj:=wPaper;
    MoveL Offs(pOrigin,241.72,63.19,6.00),vTravel,z5,tPen\WObj:=wPaper;
    MoveL Offs(pOrigin,241.72,63.19,0.00),v60,z0,tPen\WObj:=wPaper;
    MoveL Offs(pOrigin,239.76,65.14,0.00),v40,z0,tPen\WObj:=wPaper;
    MoveL Offs(pOrigin,240.29,65.85,0.00),v40,z0,tPen\WObj:=wPaper;
    MoveL Offs(pOrigin,241.49,67.06,0.00),v40,z0,tPen\WObj:=wPaper;
    MoveL Offs(pOrigin,242.15,67.23,0.00),v40,z0,tPen\WObj:=wPaper;
    MoveL Offs(pOrigin,240.20,69.18,0.00),v40,z0,tPen\WObj:=wPaper;
    MoveL Offs(pOrigin,240.90,69.45,0.00),v40,z0,tPen\WObj:=wPaper;
    MoveL Offs(pOrigin,241.65,70.20,0.00),v40,z0,tPen\WObj:=wPaper;
    MoveL Offs(pOrigin,242.30,70.08,0.00),v40,z0,tPen\WObj:=wPaper;
    MoveL Offs(pOrigin,240.34,72.03,0.00),v40,fine,tPen\WObj:=wPaper;
    MoveL Offs(pOrigin,240.34,72.03,6.00),v60,z5,tPen\WObj:=wPaper;
    MoveL Offs(pOrigin,240.90,70.95,6.00),vTravel,z5,tPen\WObj:=wPaper;
    MoveL Offs(pOrigin,240.90,70.95,0.00),v60,z0,tPen\WObj:=wPaper;
    MoveL Offs(pOrigin,241.66,71.70,0.00),v40,z0,tPen\WObj:=wPaper;
    MoveL Offs(pOrigin,242.59,71.27,0.00),v40,z0,tPen\WObj:=wPaper;
    MoveL Offs(pOrigin,240.64,73.23,0.00),v40,fine,tPen\WObj:=wPaper;
    MoveL Offs(pOrigin,240.64,73.23,6.00),v60,z5,tPen\WObj:=wPaper;
    MoveL Offs(pOrigin,241.36,74.40,6.00),vTravel,z5,tPen\WObj:=wPaper;
    MoveL Offs(pOrigin,241.36,74.40,0.00),v60,z0,tPen\WObj:=wPaper;
    MoveL Offs(pOrigin,242.12,75.15,0.00),v40,z0,tPen\WObj:=wPaper;
    MoveL Offs(pOrigin,243.03,75.32,0.00),v40,z0,tPen\WObj:=wPaper;
    MoveL Offs(pOrigin,240.92,77.42,0.00),v40,fine,tPen\WObj:=wPaper;
    MoveL Offs(pOrigin,240.92,77.42,6.00),v60,z5,tPen\WObj:=wPaper;
    MoveL Offs(pOrigin,240.78,76.07,6.00),vTravel,z5,tPen\WObj:=wPaper;
    MoveL Offs(pOrigin,240.78,76.07,0.00),v60,z0,tPen\WObj:=wPaper;
    MoveL Offs(pOrigin,242.73,74.12,0.00),v40,fine,tPen\WObj:=wPaper;
    MoveL Offs(pOrigin,242.73,74.12,6.00),v60,z5,tPen\WObj:=wPaper;
    MoveL Offs(pOrigin,242.59,72.77,6.00),vTravel,z5,tPen\WObj:=wPaper;
    MoveL Offs(pOrigin,242.59,72.77,0.00),v60,z0,tPen\WObj:=wPaper;
    MoveL Offs(pOrigin,240.63,74.73,0.00),v40,fine,tPen\WObj:=wPaper;
    MoveL Offs(pOrigin,240.63,74.73,6.00),v60,z5,tPen\WObj:=wPaper;
    MoveL Offs(pOrigin,241.37,75.89,6.00),vTravel,z5,tPen\WObj:=wPaper;
    MoveL Offs(pOrigin,241.37,75.89,0.00),v60,z0,tPen\WObj:=wPaper;
    MoveL Offs(pOrigin,242.27,76.80,0.00),v40,z0,tPen\WObj:=wPaper;
    MoveL Offs(pOrigin,243.02,76.82,0.00),v40,z0,tPen\WObj:=wPaper;
    MoveL Offs(pOrigin,240.92,78.92,0.00),v40,z0,tPen\WObj:=wPaper;
    MoveL Offs(pOrigin,241.68,79.19,0.00),v40,z0,tPen\WObj:=wPaper;
    MoveL Offs(pOrigin,242.58,80.09,0.00),v40,z0,tPen\WObj:=wPaper;
    MoveL Offs(pOrigin,243.16,79.66,0.00),v40,z0,tPen\WObj:=wPaper;
    MoveL Offs(pOrigin,241.21,81.61,0.00),v40,z0,tPen\WObj:=wPaper;
    MoveL Offs(pOrigin,241.83,80.84,0.00),v40,z0,tPen\WObj:=wPaper;
    MoveL Offs(pOrigin,242.59,81.59,0.00),v40,z0,tPen\WObj:=wPaper;
    MoveL Offs(pOrigin,243.31,81.01,0.00),v40,z0,tPen\WObj:=wPaper;
    MoveL Offs(pOrigin,241.21,83.11,0.00),v40,z0,tPen\WObj:=wPaper;
    MoveL Offs(pOrigin,241.99,83.99,0.00),v40,z0,tPen\WObj:=wPaper;
    MoveL Offs(pOrigin,242.74,84.74,0.00),v40,z0,tPen\WObj:=wPaper;
    MoveL Offs(pOrigin,243.30,84.00,0.00),v40,z0,tPen\WObj:=wPaper;
    MoveL Offs(pOrigin,241.35,85.96,0.00),v40,fine,tPen\WObj:=wPaper;
    MoveL Offs(pOrigin,241.35,85.96,6.00),v60,z5,tPen\WObj:=wPaper;
    MoveL Offs(pOrigin,241.64,87.16,6.00),vTravel,z5,tPen\WObj:=wPaper;
    MoveL Offs(pOrigin,241.64,87.16,0.00),v60,z0,tPen\WObj:=wPaper;
    MoveL Offs(pOrigin,243.60,85.20,0.00),v40,fine,tPen\WObj:=wPaper;
    MoveL Offs(pOrigin,243.60,85.20,6.00),v60,z5,tPen\WObj:=wPaper;
    MoveL Offs(pOrigin,243.59,86.70,6.00),vTravel,z5,tPen\WObj:=wPaper;
    MoveL Offs(pOrigin,243.59,86.70,0.00),v60,z0,tPen\WObj:=wPaper;
    MoveL Offs(pOrigin,241.64,88.65,0.00),v40,fine,tPen\WObj:=wPaper;
    MoveL Offs(pOrigin,241.64,88.65,6.00),v60,z5,tPen\WObj:=wPaper;
    MoveL Offs(pOrigin,241.78,90.00,6.00),vTravel,z5,tPen\WObj:=wPaper;
    MoveL Offs(pOrigin,241.78,90.00,0.00),v60,z0,tPen\WObj:=wPaper;
    MoveL Offs(pOrigin,243.74,88.05,0.00),v40,z0,tPen\WObj:=wPaper;
    MoveL Offs(pOrigin,243.05,88.03,0.00),v40,z0,tPen\WObj:=wPaper;
    MoveL Offs(pOrigin,242.30,87.28,0.00),v40,fine,tPen\WObj:=wPaper;
    MoveL Offs(pOrigin,242.30,87.28,6.00),v60,z5,tPen\WObj:=wPaper;
    MoveL Offs(pOrigin,243.73,89.55,6.00),vTravel,z5,tPen\WObj:=wPaper;
    MoveL Offs(pOrigin,243.73,89.55,0.00),v60,z0,tPen\WObj:=wPaper;
    MoveL Offs(pOrigin,241.78,91.50,0.00),v40,fine,tPen\WObj:=wPaper;
    MoveL Offs(pOrigin,241.78,91.50,6.00),v60,z5,tPen\WObj:=wPaper;
    MoveL Offs(pOrigin,242.46,90.43,6.00),vTravel,z5,tPen\WObj:=wPaper;
    MoveL Offs(pOrigin,242.46,90.43,0.00),v60,z0,tPen\WObj:=wPaper;
    MoveL Offs(pOrigin,243.21,91.18,0.00),v40,z0,tPen\WObj:=wPaper;
    MoveL Offs(pOrigin,244.03,90.74,0.00),v40,z0,tPen\WObj:=wPaper;
    MoveL Offs(pOrigin,241.78,93.00,0.00),v40,fine,tPen\WObj:=wPaper;
    MoveL Offs(pOrigin,241.78,93.00,6.00),v60,z5,tPen\WObj:=wPaper;
    MoveL Offs(pOrigin,241.92,94.35,6.00),vTravel,z5,tPen\WObj:=wPaper;
    MoveL Offs(pOrigin,241.92,94.35,0.00),v60,z0,tPen\WObj:=wPaper;
    MoveL Offs(pOrigin,244.02,92.24,0.00),v40,fine,tPen\WObj:=wPaper;
    MoveL Offs(pOrigin,244.02,92.24,6.00),v60,z5,tPen\WObj:=wPaper;
  ENDPROC

  PROC DrawPart9()
    MoveL Offs(pOrigin,244.02,93.74,6.00),vTravel,z5,tPen\WObj:=wPaper;
    MoveL Offs(pOrigin,244.02,93.74,0.00),v60,z0,tPen\WObj:=wPaper;
    MoveL Offs(pOrigin,241.92,95.84,0.00),v40,fine,tPen\WObj:=wPaper;
    MoveL Offs(pOrigin,241.92,95.84,6.00),v60,z5,tPen\WObj:=wPaper;
    MoveL Offs(pOrigin,242.21,97.04,6.00),vTravel,z5,tPen\WObj:=wPaper;
    MoveL Offs(pOrigin,242.21,97.04,0.00),v60,z0,tPen\WObj:=wPaper;
    MoveL Offs(pOrigin,244.17,95.09,0.00),v40,fine,tPen\WObj:=wPaper;
    MoveL Offs(pOrigin,244.17,95.09,6.00),v60,z5,tPen\WObj:=wPaper;
    MoveL Offs(pOrigin,244.16,96.59,6.00),vTravel,z5,tPen\WObj:=wPaper;
    MoveL Offs(pOrigin,244.16,96.59,0.00),v60,z0,tPen\WObj:=wPaper;
    MoveL Offs(pOrigin,242.21,98.54,0.00),v40,fine,tPen\WObj:=wPaper;
    MoveL Offs(pOrigin,242.21,98.54,6.00),v60,z5,tPen\WObj:=wPaper;
    MoveL Offs(pOrigin,242.35,99.89,6.00),vTravel,z5,tPen\WObj:=wPaper;
    MoveL Offs(pOrigin,242.35,99.89,0.00),v60,z0,tPen\WObj:=wPaper;
    MoveL Offs(pOrigin,244.31,97.93,0.00),v40,fine,tPen\WObj:=wPaper;
    MoveL Offs(pOrigin,244.31,97.93,6.00),v60,z5,tPen\WObj:=wPaper;
    MoveL Offs(pOrigin,244.30,99.43,6.00),vTravel,z5,tPen\WObj:=wPaper;
    MoveL Offs(pOrigin,244.30,99.43,0.00),v60,z0,tPen\WObj:=wPaper;
    MoveL Offs(pOrigin,242.35,101.38,0.00),v40,fine,tPen\WObj:=wPaper;
    MoveL Offs(pOrigin,242.35,101.38,6.00),v60,z5,tPen\WObj:=wPaper;
    MoveL Offs(pOrigin,242.34,102.88,6.00),vTravel,z5,tPen\WObj:=wPaper;
    MoveL Offs(pOrigin,242.34,102.88,0.00),v60,z0,tPen\WObj:=wPaper;
    MoveL Offs(pOrigin,244.30,100.93,0.00),v40,fine,tPen\WObj:=wPaper;
    MoveL Offs(pOrigin,244.30,100.93,6.00),v60,z5,tPen\WObj:=wPaper;
    MoveL Offs(pOrigin,244.59,102.13,6.00),vTravel,z5,tPen\WObj:=wPaper;
    MoveL Offs(pOrigin,244.59,102.13,0.00),v60,z0,tPen\WObj:=wPaper;
    MoveL Offs(pOrigin,242.34,104.38,0.00),v40,z0,tPen\WObj:=wPaper;
    MoveL Offs(pOrigin,242.79,105.43,0.00),v40,z0,tPen\WObj:=wPaper;
    MoveL Offs(pOrigin,244.74,103.47,0.00),v40,fine,tPen\WObj:=wPaper;
    MoveL Offs(pOrigin,244.74,103.47,6.00),v60,z5,tPen\WObj:=wPaper;
    MoveL Offs(pOrigin,244.73,104.97,6.00),vTravel,z5,tPen\WObj:=wPaper;
    MoveL Offs(pOrigin,244.73,104.97,0.00),v60,z0,tPen\WObj:=wPaper;
    MoveL Offs(pOrigin,242.78,106.93,0.00),v40,z0,tPen\WObj:=wPaper;
    MoveL Offs(pOrigin,243.26,106.16,0.00),v40,z0,tPen\WObj:=wPaper;
    MoveL Offs(pOrigin,244.01,106.91,0.00),v40,z0,tPen\WObj:=wPaper;
    MoveL Offs(pOrigin,244.73,106.47,0.00),v40,z0,tPen\WObj:=wPaper;
    MoveL Offs(pOrigin,242.78,108.42,0.00),v40,fine,tPen\WObj:=wPaper;
    MoveL Offs(pOrigin,242.78,108.42,6.00),v60,z5,tPen\WObj:=wPaper;
    MoveL Offs(pOrigin,242.77,109.92,6.00),vTravel,z5,tPen\WObj:=wPaper;
    MoveL Offs(pOrigin,242.77,109.92,0.00),v60,z0,tPen\WObj:=wPaper;
    MoveL Offs(pOrigin,244.88,107.82,0.00),v40,fine,tPen\WObj:=wPaper;
    MoveL Offs(pOrigin,244.88,107.82,6.00),v60,z5,tPen\WObj:=wPaper;
    MoveL Offs(pOrigin,244.87,109.32,6.00),vTravel,z5,tPen\WObj:=wPaper;
    MoveL Offs(pOrigin,244.87,109.32,0.00),v60,z0,tPen\WObj:=wPaper;
    MoveL Offs(pOrigin,242.92,111.27,0.00),v40,fine,tPen\WObj:=wPaper;
    MoveL Offs(pOrigin,242.92,111.27,6.00),v60,z5,tPen\WObj:=wPaper;
    MoveL Offs(pOrigin,242.91,112.77,6.00),vTravel,z5,tPen\WObj:=wPaper;
    MoveL Offs(pOrigin,242.91,112.77,0.00),v60,z0,tPen\WObj:=wPaper;
    MoveL Offs(pOrigin,244.87,110.81,0.00),v40,fine,tPen\WObj:=wPaper;
    MoveL Offs(pOrigin,244.87,110.81,6.00),v60,z5,tPen\WObj:=wPaper;
    MoveL Offs(pOrigin,244.86,112.31,6.00),vTravel,z5,tPen\WObj:=wPaper;
    MoveL Offs(pOrigin,244.86,112.31,0.00),v60,z0,tPen\WObj:=wPaper;
    MoveL Offs(pOrigin,242.91,114.27,0.00),v40,fine,tPen\WObj:=wPaper;
    MoveL Offs(pOrigin,242.91,114.27,6.00),v60,z5,tPen\WObj:=wPaper;
    MoveL Offs(pOrigin,242.90,115.76,6.00),vTravel,z5,tPen\WObj:=wPaper;
    MoveL Offs(pOrigin,242.90,115.76,0.00),v60,z0,tPen\WObj:=wPaper;
    MoveL Offs(pOrigin,244.86,113.81,0.00),v40,fine,tPen\WObj:=wPaper;
    MoveL Offs(pOrigin,244.86,113.81,6.00),v60,z5,tPen\WObj:=wPaper;
    MoveL Offs(pOrigin,244.85,115.31,6.00),vTravel,z5,tPen\WObj:=wPaper;
    MoveL Offs(pOrigin,244.85,115.31,0.00),v60,z0,tPen\WObj:=wPaper;
    MoveL Offs(pOrigin,242.90,117.26,0.00),v40,fine,tPen\WObj:=wPaper;
    MoveL Offs(pOrigin,242.90,117.26,6.00),v60,z5,tPen\WObj:=wPaper;
    MoveL Offs(pOrigin,243.04,118.61,6.00),vTravel,z5,tPen\WObj:=wPaper;
    MoveL Offs(pOrigin,243.04,118.61,0.00),v60,z0,tPen\WObj:=wPaper;
    MoveL Offs(pOrigin,245.15,116.51,0.00),v40,fine,tPen\WObj:=wPaper;
    MoveL Offs(pOrigin,245.15,116.51,6.00),v60,z5,tPen\WObj:=wPaper;
    MoveL Offs(pOrigin,245.14,118.00,6.00),vTravel,z5,tPen\WObj:=wPaper;
    MoveL Offs(pOrigin,245.14,118.00,0.00),v60,z0,tPen\WObj:=wPaper;
    MoveL Offs(pOrigin,243.19,119.96,0.00),v40,fine,tPen\WObj:=wPaper;
    MoveL Offs(pOrigin,243.19,119.96,6.00),v60,z5,tPen\WObj:=wPaper;
    MoveL Offs(pOrigin,243.19,121.46,6.00),vTravel,z5,tPen\WObj:=wPaper;
    MoveL Offs(pOrigin,243.19,121.46,0.00),v60,z0,tPen\WObj:=wPaper;
    MoveL Offs(pOrigin,245.14,119.50,0.00),v40,fine,tPen\WObj:=wPaper;
    MoveL Offs(pOrigin,245.14,119.50,6.00),v60,z5,tPen\WObj:=wPaper;
    MoveL Offs(pOrigin,245.13,121.00,6.00),vTravel,z5,tPen\WObj:=wPaper;
    MoveL Offs(pOrigin,245.13,121.00,0.00),v60,z0,tPen\WObj:=wPaper;
    MoveL Offs(pOrigin,243.18,122.95,0.00),v40,fine,tPen\WObj:=wPaper;
    MoveL Offs(pOrigin,243.18,122.95,6.00),v60,z5,tPen\WObj:=wPaper;
    MoveL Offs(pOrigin,243.18,124.45,6.00),vTravel,z5,tPen\WObj:=wPaper;
    MoveL Offs(pOrigin,243.18,124.45,0.00),v60,z0,tPen\WObj:=wPaper;
    MoveL Offs(pOrigin,245.28,122.35,0.00),v40,fine,tPen\WObj:=wPaper;
    MoveL Offs(pOrigin,245.28,122.35,6.00),v60,z5,tPen\WObj:=wPaper;
    MoveL Offs(pOrigin,245.28,123.85,6.00),vTravel,z5,tPen\WObj:=wPaper;
    MoveL Offs(pOrigin,245.28,123.85,0.00),v60,z0,tPen\WObj:=wPaper;
    MoveL Offs(pOrigin,243.17,125.95,0.00),v40,fine,tPen\WObj:=wPaper;
    MoveL Offs(pOrigin,243.17,125.95,6.00),v60,z5,tPen\WObj:=wPaper;
    MoveL Offs(pOrigin,243.17,127.45,6.00),vTravel,z5,tPen\WObj:=wPaper;
    MoveL Offs(pOrigin,243.17,127.45,0.00),v60,z0,tPen\WObj:=wPaper;
    MoveL Offs(pOrigin,245.27,125.34,0.00),v40,fine,tPen\WObj:=wPaper;
    MoveL Offs(pOrigin,245.27,125.34,6.00),v60,z5,tPen\WObj:=wPaper;
    MoveL Offs(pOrigin,245.27,126.84,6.00),vTravel,z5,tPen\WObj:=wPaper;
    MoveL Offs(pOrigin,245.27,126.84,0.00),v60,z0,tPen\WObj:=wPaper;
    MoveL Offs(pOrigin,243.31,128.79,0.00),v40,fine,tPen\WObj:=wPaper;
    MoveL Offs(pOrigin,243.31,128.79,6.00),v60,z5,tPen\WObj:=wPaper;
    MoveL Offs(pOrigin,243.31,130.29,6.00),vTravel,z5,tPen\WObj:=wPaper;
    MoveL Offs(pOrigin,243.31,130.29,0.00),v60,z0,tPen\WObj:=wPaper;
    MoveL Offs(pOrigin,245.26,128.34,0.00),v40,fine,tPen\WObj:=wPaper;
    MoveL Offs(pOrigin,245.26,128.34,6.00),v60,z5,tPen\WObj:=wPaper;
    MoveL Offs(pOrigin,245.41,129.69,6.00),vTravel,z5,tPen\WObj:=wPaper;
    MoveL Offs(pOrigin,245.41,129.69,0.00),v60,z0,tPen\WObj:=wPaper;
    MoveL Offs(pOrigin,243.30,131.79,0.00),v40,fine,tPen\WObj:=wPaper;
    MoveL Offs(pOrigin,243.30,131.79,6.00),v60,z5,tPen\WObj:=wPaper;
    MoveL Offs(pOrigin,243.30,133.29,6.00),vTravel,z5,tPen\WObj:=wPaper;
    MoveL Offs(pOrigin,243.30,133.29,0.00),v60,z0,tPen\WObj:=wPaper;
    MoveL Offs(pOrigin,245.55,131.03,0.00),v40,fine,tPen\WObj:=wPaper;
    MoveL Offs(pOrigin,245.55,131.03,6.00),v60,z5,tPen\WObj:=wPaper;
    MoveL Offs(pOrigin,245.55,132.53,6.00),vTravel,z5,tPen\WObj:=wPaper;
    MoveL Offs(pOrigin,245.55,132.53,0.00),v60,z0,tPen\WObj:=wPaper;
    MoveL Offs(pOrigin,243.29,134.79,0.00),v40,fine,tPen\WObj:=wPaper;
    MoveL Offs(pOrigin,243.29,134.79,6.00),v60,z5,tPen\WObj:=wPaper;
    MoveL Offs(pOrigin,244.25,135.52,6.00),vTravel,z5,tPen\WObj:=wPaper;
    MoveL Offs(pOrigin,244.25,135.52,0.00),v60,z0,tPen\WObj:=wPaper;
    MoveL Offs(pOrigin,245.15,136.42,0.00),v40,z0,tPen\WObj:=wPaper;
    MoveL Offs(pOrigin,245.69,136.88,0.00),v40,z0,tPen\WObj:=wPaper;
    MoveL Offs(pOrigin,243.43,139.13,0.00),v40,z0,tPen\WObj:=wPaper;
    MoveL Offs(pOrigin,244.26,138.52,0.00),v40,z0,tPen\WObj:=wPaper;
    MoveL Offs(pOrigin,245.31,139.57,0.00),v40,z0,tPen\WObj:=wPaper;
    MoveL Offs(pOrigin,245.83,139.72,0.00),v40,z0,tPen\WObj:=wPaper;
    MoveL Offs(pOrigin,243.72,141.83,0.00),v40,z0,tPen\WObj:=wPaper;
    MoveL Offs(pOrigin,244.42,141.67,0.00),v40,z0,tPen\WObj:=wPaper;
  ENDPROC

  PROC DrawPart10()
    MoveL Offs(pOrigin,245.62,142.87,0.00),v40,z0,tPen\WObj:=wPaper;
    MoveL Offs(pOrigin,246.12,142.42,0.00),v40,z0,tPen\WObj:=wPaper;
    MoveL Offs(pOrigin,243.86,144.67,0.00),v40,z0,tPen\WObj:=wPaper;
    MoveL Offs(pOrigin,244.58,144.81,0.00),v40,z0,tPen\WObj:=wPaper;
    MoveL Offs(pOrigin,245.78,146.01,0.00),v40,z0,tPen\WObj:=wPaper;
    MoveL Offs(pOrigin,245.11,145.68,0.00),v40,z0,tPen\WObj:=wPaper;
    MoveL Offs(pOrigin,244.90,146.74,0.00),v40,z0,tPen\WObj:=wPaper;
    MoveL Offs(pOrigin,245.32,147.16,0.00),v40,z0,tPen\WObj:=wPaper;
    MoveL Offs(pOrigin,245.32,147.59,0.00),v40,z0,tPen\WObj:=wPaper;
    MoveL Offs(pOrigin,245.75,146.31,0.00),v40,z0,tPen\WObj:=wPaper;
    MoveL Offs(pOrigin,245.11,145.25,0.00),v40,z0,tPen\WObj:=wPaper;
    MoveL Offs(pOrigin,245.54,144.40,0.00),v40,z0,tPen\WObj:=wPaper;
    MoveL Offs(pOrigin,244.90,142.91,0.00),v40,z0,tPen\WObj:=wPaper;
    MoveL Offs(pOrigin,245.32,141.43,0.00),v40,z0,tPen\WObj:=wPaper;
    MoveL Offs(pOrigin,244.69,140.36,0.00),v40,z0,tPen\WObj:=wPaper;
    MoveL Offs(pOrigin,244.69,138.66,0.00),v40,z0,tPen\WObj:=wPaper;
    MoveL Offs(pOrigin,245.11,137.60,0.00),v40,z0,tPen\WObj:=wPaper;
    MoveL Offs(pOrigin,244.48,136.54,0.00),v40,z0,tPen\WObj:=wPaper;
    MoveL Offs(pOrigin,243.41,97.86,0.00),v40,z0,tPen\WObj:=wPaper;
    MoveL Offs(pOrigin,241.93,75.76,0.00),v40,z0,tPen\WObj:=wPaper;
    MoveL Offs(pOrigin,239.38,51.54,0.00),v40,z0,tPen\WObj:=wPaper;
    MoveL Offs(pOrigin,238.74,40.91,0.00),v40,z0,tPen\WObj:=wPaper;
    MoveL Offs(pOrigin,238.74,40.91,0.00),v40,z0,tPen\WObj:=wPaper;
    MoveL Offs(pOrigin,239.16,40.49,0.00),v40,z0,tPen\WObj:=wPaper;
    MoveL Offs(pOrigin,240.65,40.28,0.00),v40,z0,tPen\WObj:=wPaper;
    MoveL Offs(pOrigin,242.35,40.49,0.00),v40,z0,tPen\WObj:=wPaper;
    MoveL Offs(pOrigin,245.75,45.16,0.00),v40,z0,tPen\WObj:=wPaper;
    MoveL Offs(pOrigin,254.46,54.30,0.00),v40,z0,tPen\WObj:=wPaper;
    MoveL Offs(pOrigin,254.89,55.36,0.00),v40,z0,tPen\WObj:=wPaper;
    MoveL Offs(pOrigin,254.89,55.36,0.00),v40,z0,tPen\WObj:=wPaper;
    MoveL Offs(pOrigin,257.44,79.80,0.00),v40,z0,tPen\WObj:=wPaper;
    MoveL Offs(pOrigin,258.08,89.36,0.00),v40,z0,tPen\WObj:=wPaper;
    MoveL Offs(pOrigin,258.08,89.36,0.00),v40,z0,tPen\WObj:=wPaper;
    MoveL Offs(pOrigin,258.50,89.57,0.00),v40,z0,tPen\WObj:=wPaper;
    MoveL Offs(pOrigin,258.50,90.43,0.00),v40,z0,tPen\WObj:=wPaper;
    MoveL Offs(pOrigin,257.86,90.64,0.00),v40,z0,tPen\WObj:=wPaper;
    MoveL Offs(pOrigin,257.86,90.64,0.00),v40,z0,tPen\WObj:=wPaper;
    MoveL Offs(pOrigin,258.92,94.04,0.00),v40,z0,tPen\WObj:=wPaper;
    MoveL Offs(pOrigin,258.92,94.04,0.00),v40,z0,tPen\WObj:=wPaper;
    MoveL Offs(pOrigin,260.06,95.10,0.00),v40,z0,tPen\WObj:=wPaper;
    MoveL Offs(pOrigin,263.67,102.54,0.00),v40,z0,tPen\WObj:=wPaper;
    MoveL Offs(pOrigin,269.34,116.78,0.00),v40,z0,tPen\WObj:=wPaper;
    MoveL Offs(pOrigin,269.12,116.43,0.00),v40,z0,tPen\WObj:=wPaper;
    MoveL Offs(pOrigin,272.87,112.68,0.00),v40,z0,tPen\WObj:=wPaper;
    MoveL Offs(pOrigin,272.34,112.84,0.00),v40,z0,tPen\WObj:=wPaper;
    MoveL Offs(pOrigin,270.09,110.59,0.00),v40,z0,tPen\WObj:=wPaper;
    MoveL Offs(pOrigin,270.61,110.04,0.00),v40,z0,tPen\WObj:=wPaper;
    MoveL Offs(pOrigin,271.68,110.04,0.00),v40,z0,tPen\WObj:=wPaper;
    MoveL Offs(pOrigin,272.33,109.84,0.00),v40,z0,tPen\WObj:=wPaper;
    MoveL Offs(pOrigin,269.93,107.44,0.00),v40,z0,tPen\WObj:=wPaper;
    MoveL Offs(pOrigin,269.44,107.14,0.00),v40,z0,tPen\WObj:=wPaper;
    MoveL Offs(pOrigin,272.75,103.84,0.00),v40,z0,tPen\WObj:=wPaper;
    MoveL Offs(pOrigin,272.31,103.85,0.00),v40,z0,tPen\WObj:=wPaper;
    MoveL Offs(pOrigin,269.91,101.45,0.00),v40,z0,tPen\WObj:=wPaper;
    MoveL Offs(pOrigin,269.46,101.15,0.00),v40,z0,tPen\WObj:=wPaper;
    MoveL Offs(pOrigin,272.92,97.70,0.00),v40,z0,tPen\WObj:=wPaper;
    MoveL Offs(pOrigin,272.45,98.01,0.00),v40,z0,tPen\WObj:=wPaper;
    MoveL Offs(pOrigin,270.34,95.91,0.00),v40,z0,tPen\WObj:=wPaper;
    MoveL Offs(pOrigin,270.82,96.31,0.00),v40,z0,tPen\WObj:=wPaper;
    MoveL Offs(pOrigin,271.89,96.31,0.00),v40,z0,tPen\WObj:=wPaper;
    MoveL Offs(pOrigin,272.44,96.51,0.00),v40,z0,tPen\WObj:=wPaper;
    MoveL Offs(pOrigin,270.34,94.41,0.00),v40,z0,tPen\WObj:=wPaper;
    MoveL Offs(pOrigin,271.04,94.20,0.00),v40,z0,tPen\WObj:=wPaper;
    MoveL Offs(pOrigin,272.10,94.20,0.00),v40,z0,tPen\WObj:=wPaper;
    MoveL Offs(pOrigin,272.73,93.82,0.00),v40,z0,tPen\WObj:=wPaper;
    MoveL Offs(pOrigin,270.48,91.56,0.00),v40,z0,tPen\WObj:=wPaper;
    MoveL Offs(pOrigin,269.94,91.71,0.00),v40,z0,tPen\WObj:=wPaper;
    MoveL Offs(pOrigin,273.85,87.81,0.00),v40,z0,tPen\WObj:=wPaper;
    MoveL Offs(pOrigin,273.01,88.12,0.00),v40,z0,tPen\WObj:=wPaper;
    MoveL Offs(pOrigin,270.91,86.02,0.00),v40,z0,tPen\WObj:=wPaper;
    MoveL Offs(pOrigin,270.56,86.62,0.00),v40,z0,tPen\WObj:=wPaper;
    MoveL Offs(pOrigin,274.16,83.01,0.00),v40,z0,tPen\WObj:=wPaper;
    MoveL Offs(pOrigin,273.75,82.88,0.00),v40,z0,tPen\WObj:=wPaper;
    MoveL Offs(pOrigin,270.89,80.03,0.00),v40,z0,tPen\WObj:=wPaper;
    MoveL Offs(pOrigin,270.57,80.63,0.00),v40,z0,tPen\WObj:=wPaper;
    MoveL Offs(pOrigin,275.23,75.97,0.00),v40,z0,tPen\WObj:=wPaper;
    MoveL Offs(pOrigin,274.63,76.30,0.00),v40,z0,tPen\WObj:=wPaper;
    MoveL Offs(pOrigin,272.52,74.19,0.00),v40,z0,tPen\WObj:=wPaper;
    MoveL Offs(pOrigin,273.16,74.14,0.00),v40,z0,tPen\WObj:=wPaper;
    MoveL Offs(pOrigin,274.44,74.14,0.00),v40,z0,tPen\WObj:=wPaper;
    MoveL Offs(pOrigin,275.07,73.75,0.00),v40,z0,tPen\WObj:=wPaper;
    MoveL Offs(pOrigin,272.96,71.65,0.00),v40,z0,tPen\WObj:=wPaper;
    MoveL Offs(pOrigin,272.40,71.33,0.00),v40,z0,tPen\WObj:=wPaper;
    MoveL Offs(pOrigin,278.71,65.02,0.00),v40,z0,tPen\WObj:=wPaper;
    MoveL Offs(pOrigin,279.09,65.82,0.00),v40,z0,tPen\WObj:=wPaper;
    MoveL Offs(pOrigin,282.09,68.83,0.00),v40,z0,tPen\WObj:=wPaper;
    MoveL Offs(pOrigin,281.84,69.36,0.00),v40,z0,tPen\WObj:=wPaper;
    MoveL Offs(pOrigin,285.90,65.30,0.00),v40,z0,tPen\WObj:=wPaper;
    MoveL Offs(pOrigin,286.58,65.85,0.00),v40,z0,tPen\WObj:=wPaper;
    MoveL Offs(pOrigin,288.08,67.35,0.00),v40,z0,tPen\WObj:=wPaper;
    MoveL Offs(pOrigin,288.04,66.74,0.00),v40,z0,tPen\WObj:=wPaper;
    MoveL Offs(pOrigin,285.27,66.74,0.00),v40,z0,tPen\WObj:=wPaper;
    MoveL Offs(pOrigin,285.53,66.29,0.00),v40,z0,tPen\WObj:=wPaper;
    MoveL Offs(pOrigin,287.18,67.95,0.00),v40,z0,tPen\WObj:=wPaper;
    MoveL Offs(pOrigin,286.76,67.80,0.00),v40,z0,tPen\WObj:=wPaper;
    MoveL Offs(pOrigin,280.18,67.80,0.00),v40,z0,tPen\WObj:=wPaper;
    MoveL Offs(pOrigin,280.44,68.67,0.00),v40,z0,tPen\WObj:=wPaper;
    MoveL Offs(pOrigin,276.24,64.47,0.00),v40,z0,tPen\WObj:=wPaper;
    MoveL Offs(pOrigin,276.62,64.13,0.00),v40,z0,tPen\WObj:=wPaper;
    MoveL Offs(pOrigin,273.01,67.74,0.00),v40,z0,tPen\WObj:=wPaper;
    MoveL Offs(pOrigin,273.70,67.90,0.00),v40,z0,tPen\WObj:=wPaper;
    MoveL Offs(pOrigin,275.65,69.86,0.00),v40,z0,tPen\WObj:=wPaper;
    MoveL Offs(pOrigin,275.08,69.91,0.00),v40,z0,tPen\WObj:=wPaper;
    MoveL Offs(pOrigin,273.80,69.91,0.00),v40,z0,tPen\WObj:=wPaper;
    MoveL Offs(pOrigin,273.56,69.25,0.00),v40,z0,tPen\WObj:=wPaper;
    MoveL Offs(pOrigin,275.51,71.21,0.00),v40,z0,tPen\WObj:=wPaper;
    MoveL Offs(pOrigin,275.08,70.97,0.00),v40,z0,tPen\WObj:=wPaper;
    MoveL Offs(pOrigin,273.59,70.97,0.00),v40,z0,tPen\WObj:=wPaper;
    MoveL Offs(pOrigin,273.26,70.45,0.00),v40,z0,tPen\WObj:=wPaper;
    MoveL Offs(pOrigin,275.21,72.40,0.00),v40,z0,tPen\WObj:=wPaper;
    MoveL Offs(pOrigin,274.86,72.02,0.00),v40,z0,tPen\WObj:=wPaper;
    MoveL Offs(pOrigin,273.59,72.02,0.00),v40,z0,tPen\WObj:=wPaper;
    MoveL Offs(pOrigin,273.38,73.08,0.00),v40,z0,tPen\WObj:=wPaper;
    MoveL Offs(pOrigin,274.65,73.08,0.00),v40,fine,tPen\WObj:=wPaper;
    MoveL Offs(pOrigin,274.65,73.08,6.00),v60,z5,tPen\WObj:=wPaper;
    MoveL Offs(pOrigin,275.54,74.17,6.00),vTravel,z5,tPen\WObj:=wPaper;
    MoveL Offs(pOrigin,275.54,74.17,0.00),v60,z0,tPen\WObj:=wPaper;
    MoveL Offs(pOrigin,270.13,79.58,0.00),v40,z0,tPen\WObj:=wPaper;
    MoveL Offs(pOrigin,269.68,78.53,0.00),v40,z0,tPen\WObj:=wPaper;
    MoveL Offs(pOrigin,275.99,72.22,0.00),v40,fine,tPen\WObj:=wPaper;
  ENDPROC

  PROC DrawPart11()
    MoveL Offs(pOrigin,275.99,72.22,6.00),v60,z5,tPen\WObj:=wPaper;
    MoveL Offs(pOrigin,276.00,70.72,6.00),vTravel,z5,tPen\WObj:=wPaper;
    MoveL Offs(pOrigin,276.00,70.72,0.00),v60,z0,tPen\WObj:=wPaper;
    MoveL Offs(pOrigin,271.64,75.08,0.00),v40,z0,tPen\WObj:=wPaper;
    MoveL Offs(pOrigin,272.53,75.69,0.00),v40,z0,tPen\WObj:=wPaper;
    MoveL Offs(pOrigin,274.48,77.64,0.00),v40,z0,tPen\WObj:=wPaper;
    MoveL Offs(pOrigin,274.01,77.30,0.00),v40,z0,tPen\WObj:=wPaper;
    MoveL Offs(pOrigin,272.74,77.30,0.00),v40,z0,tPen\WObj:=wPaper;
    MoveL Offs(pOrigin,272.08,76.74,0.00),v40,z0,tPen\WObj:=wPaper;
    MoveL Offs(pOrigin,274.18,78.84,0.00),v40,z0,tPen\WObj:=wPaper;
    MoveL Offs(pOrigin,273.80,78.36,0.00),v40,z0,tPen\WObj:=wPaper;
    MoveL Offs(pOrigin,272.31,78.36,0.00),v40,z0,tPen\WObj:=wPaper;
    MoveL Offs(pOrigin,271.63,77.78,0.00),v40,z0,tPen\WObj:=wPaper;
    MoveL Offs(pOrigin,274.04,80.19,0.00),v40,z0,tPen\WObj:=wPaper;
    MoveL Offs(pOrigin,273.59,80.47,0.00),v40,z0,tPen\WObj:=wPaper;
    MoveL Offs(pOrigin,271.89,80.47,0.00),v40,z0,tPen\WObj:=wPaper;
    MoveL Offs(pOrigin,271.67,79.59,0.00),v40,z0,tPen\WObj:=wPaper;
    MoveL Offs(pOrigin,272.10,79.38,0.00),v40,z0,tPen\WObj:=wPaper;
    MoveL Offs(pOrigin,272.52,78.31,0.00),v40,z0,tPen\WObj:=wPaper;
    MoveL Offs(pOrigin,273.38,71.72,0.00),v40,z0,tPen\WObj:=wPaper;
    MoveL Offs(pOrigin,274.44,66.84,0.00),v40,z0,tPen\WObj:=wPaper;
    MoveL Offs(pOrigin,274.37,65.78,0.00),v40,z0,tPen\WObj:=wPaper;
    MoveL Offs(pOrigin,271.04,64.00,0.00),v40,z0,tPen\WObj:=wPaper;
    MoveL Offs(pOrigin,261.69,60.11,0.00),v40,z0,tPen\WObj:=wPaper;
    MoveL Offs(pOrigin,258.29,57.91,0.00),v40,z0,tPen\WObj:=wPaper;
    MoveL Offs(pOrigin,255.95,55.79,0.00),v40,z0,tPen\WObj:=wPaper;
    MoveL Offs(pOrigin,254.89,55.36,0.00),v40,z0,tPen\WObj:=wPaper;
    MoveL Offs(pOrigin,255.31,55.13,0.00),v40,z0,tPen\WObj:=wPaper;
    MoveL Offs(pOrigin,257.23,55.13,0.00),v40,z0,tPen\WObj:=wPaper;
    MoveL Offs(pOrigin,257.44,55.36,0.00),v40,z0,tPen\WObj:=wPaper;
    MoveL Offs(pOrigin,258.08,56.00,0.00),v40,z0,tPen\WObj:=wPaper;
    MoveL Offs(pOrigin,257.44,55.36,0.00),v40,z0,tPen\WObj:=wPaper;
    MoveL Offs(pOrigin,257.48,54.67,0.00),v40,z0,tPen\WObj:=wPaper;
    MoveL Offs(pOrigin,264.85,62.03,0.00),v40,z0,tPen\WObj:=wPaper;
    MoveL Offs(pOrigin,264.79,62.52,0.00),v40,z0,tPen\WObj:=wPaper;
    MoveL Offs(pOrigin,273.80,53.50,0.00),v40,z0,tPen\WObj:=wPaper;
    MoveL Offs(pOrigin,273.36,54.12,0.00),v40,z0,tPen\WObj:=wPaper;
    MoveL Offs(pOrigin,276.21,56.98,0.00),v40,z0,tPen\WObj:=wPaper;
    MoveL Offs(pOrigin,276.04,57.24,0.00),v40,z0,tPen\WObj:=wPaper;
    MoveL Offs(pOrigin,278.14,55.14,0.00),v40,z0,tPen\WObj:=wPaper;
    MoveL Offs(pOrigin,278.01,55.78,0.00),v40,z0,tPen\WObj:=wPaper;
    MoveL Offs(pOrigin,280.86,58.64,0.00),v40,z0,tPen\WObj:=wPaper;
    MoveL Offs(pOrigin,280.23,59.02,0.00),v40,z0,tPen\WObj:=wPaper;
    MoveL Offs(pOrigin,281.73,57.52,0.00),v40,z0,tPen\WObj:=wPaper;
    MoveL Offs(pOrigin,282.48,58.27,0.00),v40,z0,tPen\WObj:=wPaper;
    MoveL Offs(pOrigin,281.28,59.47,0.00),v40,fine,tPen\WObj:=wPaper;
    MoveL Offs(pOrigin,281.28,59.47,6.00),v60,z5,tPen\WObj:=wPaper;
    MoveL Offs(pOrigin,283.15,60.46,6.00),vTravel,z5,tPen\WObj:=wPaper;
    MoveL Offs(pOrigin,283.15,60.46,0.00),v60,z0,tPen\WObj:=wPaper;
    MoveL Offs(pOrigin,281.66,58.83,0.00),v40,z0,tPen\WObj:=wPaper;
    MoveL Offs(pOrigin,279.96,57.70,0.00),v40,z0,tPen\WObj:=wPaper;
    MoveL Offs(pOrigin,279.96,57.70,0.00),v40,z0,tPen\WObj:=wPaper;
    MoveL Offs(pOrigin,279.54,56.92,0.00),v40,z0,tPen\WObj:=wPaper;
    MoveL Offs(pOrigin,278.48,56.28,0.00),v40,z0,tPen\WObj:=wPaper;
    MoveL Offs(pOrigin,269.34,52.88,0.00),v40,z0,tPen\WObj:=wPaper;
    MoveL Offs(pOrigin,265.30,50.97,0.00),v40,z0,tPen\WObj:=wPaper;
    MoveL Offs(pOrigin,259.35,47.08,0.00),v40,z0,tPen\WObj:=wPaper;
    MoveL Offs(pOrigin,250.21,40.28,0.00),v40,z0,tPen\WObj:=wPaper;
    MoveL Offs(pOrigin,248.80,39.00,0.00),v40,z0,tPen\WObj:=wPaper;
    MoveL Offs(pOrigin,248.30,37.94,0.00),v40,z0,tPen\WObj:=wPaper;
    MoveL Offs(pOrigin,245.82,35.95,0.00),v40,z0,tPen\WObj:=wPaper;
    MoveL Offs(pOrigin,245.32,34.75,0.00),v40,z0,tPen\WObj:=wPaper;
    MoveL Offs(pOrigin,245.54,32.84,0.00),v40,z0,tPen\WObj:=wPaper;
    MoveL Offs(pOrigin,246.39,31.63,0.00),v40,z0,tPen\WObj:=wPaper;
    MoveL Offs(pOrigin,247.66,31.14,0.00),v40,z0,tPen\WObj:=wPaper;
    MoveL Offs(pOrigin,250.00,31.56,0.00),v40,z0,tPen\WObj:=wPaper;
    MoveL Offs(pOrigin,250.00,31.56,0.00),v40,z0,tPen\WObj:=wPaper;
    MoveL Offs(pOrigin,251.06,31.35,0.00),v40,z0,tPen\WObj:=wPaper;
    MoveL Offs(pOrigin,253.19,32.34,0.00),v40,z0,tPen\WObj:=wPaper;
    MoveL Offs(pOrigin,259.35,36.52,0.00),v40,z0,tPen\WObj:=wPaper;
    MoveL Offs(pOrigin,274.86,44.17,0.00),v40,z0,tPen\WObj:=wPaper;
    MoveL Offs(pOrigin,287.40,48.78,0.00),v40,z0,tPen\WObj:=wPaper;
    MoveL Offs(pOrigin,288.89,48.56,0.00),v40,z0,tPen\WObj:=wPaper;
    MoveL Offs(pOrigin,290.16,48.99,0.00),v40,z0,tPen\WObj:=wPaper;
    MoveL Offs(pOrigin,289.40,48.36,0.00),v40,z0,tPen\WObj:=wPaper;
    MoveL Offs(pOrigin,288.20,49.56,0.00),v40,z0,tPen\WObj:=wPaper;
    MoveL Offs(pOrigin,287.57,48.92,0.00),v40,z0,tPen\WObj:=wPaper;
    MoveL Offs(pOrigin,282.92,44.26,0.00),v40,z0,tPen\WObj:=wPaper;
    MoveL Offs(pOrigin,283.15,44.57,0.00),v40,z0,tPen\WObj:=wPaper;
    MoveL Offs(pOrigin,284.42,44.57,0.00),v40,z0,tPen\WObj:=wPaper;
    MoveL Offs(pOrigin,284.21,44.74,0.00),v40,z0,tPen\WObj:=wPaper;
    MoveL Offs(pOrigin,284.21,43.25,0.00),v40,z0,tPen\WObj:=wPaper;
    MoveL Offs(pOrigin,284.21,43.25,0.00),v40,z0,tPen\WObj:=wPaper;
    MoveL Offs(pOrigin,285.06,42.68,0.00),v40,z0,tPen\WObj:=wPaper;
    MoveL Offs(pOrigin,286.12,43.96,0.00),v40,z0,tPen\WObj:=wPaper;
    MoveL Offs(pOrigin,288.67,44.67,0.00),v40,z0,tPen\WObj:=wPaper;
    MoveL Offs(pOrigin,289.31,44.45,0.00),v40,z0,tPen\WObj:=wPaper;
    MoveL Offs(pOrigin,289.52,44.74,0.00),v40,z0,tPen\WObj:=wPaper;
    MoveL Offs(pOrigin,289.31,45.80,0.00),v40,z0,tPen\WObj:=wPaper;
    MoveL Offs(pOrigin,289.31,45.80,0.00),v40,z0,tPen\WObj:=wPaper;
    MoveL Offs(pOrigin,288.89,46.58,0.00),v40,z0,tPen\WObj:=wPaper;
    MoveL Offs(pOrigin,287.61,46.65,0.00),v40,z0,tPen\WObj:=wPaper;
    MoveL Offs(pOrigin,286.83,47.08,0.00),v40,z0,tPen\WObj:=wPaper;
    MoveL Offs(pOrigin,288.04,48.56,0.00),v40,z0,tPen\WObj:=wPaper;
    MoveL Offs(pOrigin,288.17,48.03,0.00),v40,z0,tPen\WObj:=wPaper;
    MoveL Offs(pOrigin,283.36,43.22,0.00),v40,z0,tPen\WObj:=wPaper;
    MoveL Offs(pOrigin,284.21,43.25,0.00),v40,z0,tPen\WObj:=wPaper;
    MoveL Offs(pOrigin,283.36,43.67,0.00),v40,z0,tPen\WObj:=wPaper;
    MoveL Offs(pOrigin,283.15,45.16,0.00),v40,z0,tPen\WObj:=wPaper;
    MoveL Offs(pOrigin,283.15,45.16,0.00),v40,z0,tPen\WObj:=wPaper;
    MoveL Offs(pOrigin,284.21,45.16,0.00),v40,z0,tPen\WObj:=wPaper;
    MoveL Offs(pOrigin,284.21,45.16,0.00),v40,z0,tPen\WObj:=wPaper;
    MoveL Offs(pOrigin,284.42,46.22,0.00),v40,z0,tPen\WObj:=wPaper;
    MoveL Offs(pOrigin,284.42,45.80,0.00),v40,z0,tPen\WObj:=wPaper;
    MoveL Offs(pOrigin,285.49,45.59,0.00),v40,z0,tPen\WObj:=wPaper;
    MoveL Offs(pOrigin,285.49,45.59,0.00),v40,z0,tPen\WObj:=wPaper;
    MoveL Offs(pOrigin,285.06,44.74,0.00),v40,z0,tPen\WObj:=wPaper;
    MoveL Offs(pOrigin,284.21,44.74,0.00),v40,fine,tPen\WObj:=wPaper;
    MoveL Offs(pOrigin,284.21,44.74,6.00),v60,z5,tPen\WObj:=wPaper;
    MoveL Offs(pOrigin,285.91,46.01,6.00),vTravel,z5,tPen\WObj:=wPaper;
    MoveL Offs(pOrigin,285.91,46.01,0.00),v60,z0,tPen\WObj:=wPaper;
    MoveL Offs(pOrigin,285.27,46.44,0.00),v40,z0,tPen\WObj:=wPaper;
    MoveL Offs(pOrigin,283.58,46.22,0.00),v40,z0,tPen\WObj:=wPaper;
    MoveL Offs(pOrigin,282.73,45.23,0.00),v40,z0,tPen\WObj:=wPaper;
    MoveL Offs(pOrigin,280.81,45.16,0.00),v40,z0,tPen\WObj:=wPaper;
    MoveL Offs(pOrigin,275.92,43.32,0.00),v40,z0,tPen\WObj:=wPaper;
    MoveL Offs(pOrigin,259.14,35.03,0.00),v40,z0,tPen\WObj:=wPaper;
    MoveL Offs(pOrigin,258.57,34.54,0.00),v40,z0,tPen\WObj:=wPaper;
    MoveL Offs(pOrigin,258.50,33.90,0.00),v40,z0,tPen\WObj:=wPaper;
    MoveL Offs(pOrigin,258.50,33.90,0.00),v40,z0,tPen\WObj:=wPaper;
  ENDPROC

